(* CODESYS project ProjectX3_HLD.project

Project tree, tasks and I/O mapping:
  Device : CODESYS Control Win V3, 3S - Smart Software Solutions GmbH, version 3.5.16.20
    application Application
      libraries: Standard, * (System)
      task MainTask (cyclic, interval 20 ms, priority 1) calls Simulation, GAinstances, POLICY
      task VISU_TASK (cyclic, interval 100 ms, priority 31) calls VisuElems.Visu_Prg
      global variables GVL
      visualisation Visualization
      program Simulation [ST]
      function block DoorGA [SFC]: Init_active, READY_active, BUSY_active, Opening_active, Opening_exit, DONE1_active, Closing_active, Closing_exit, DONE_active, RESETDONE_active, Step1_active, Openit_exit, WAIT_1_exit, EverythingGood_active, OK_comunication_active, Init_timer_active, Comun_Problem_active
      function block CalculationGA [SFC]: READY_active, BUSY_active, Init_active, Current_active, Destination_active, VariableSet_active, VariableSet2_active, DoubleOutput_active, VariableSet_exit, DeckFault_active
      program POLICY [SFC]: Motor_ON_active, Motor_OFF_active, Velocity_I_exit, Motor_OFF_exit, Door_Open_active, Door_Open_exit, Door_Close_I_active, Door_Close_exit, Array_active, led_active, DeleteArray_active, Trans6, CalculationGA_active, MotorGA_exit, Velocity_I_active, Velocity_active, Calc_I_active, MotorGA_active, Init_active, Calc_I_exit, HLD_active, OK_comunication_2_active
      function block MotorGA [SFC]: motorON_active, motorOFF_active, BUSY_active, Trans0, READY_active, Motor_ON_I_active, Motor_OFF_I_active, Trans2, Init_active, DONE1_active, DONE2_active, DONE_active, RESETDONE_active
      function block VelocityGA [SFC]: Double_Output_active, MotorSlow_active, MotorSlow_exit, MotorFast_active, StopORGo_active, RampRange_active, Init_active, READY_active, BUSY_active, Vel_Init_active, Vel_Init_exit, Ramp_Fault_active
      program GAinstances [FBD]
  text list GlobalTextList
*)

// Device/Application/GVL
{attribute 'qualified_only'}
VAR_GLOBAL
	counting:INT;
	
(* Elevator managing variables*)
	Open: BOOL;				(* Sensor: the door is fully open*)
	Closed: BOOL;			(* Sensor: the door is fully closed*)
	LimitDown: BOOL;		(* Sensor: lower limit sensor, if TRUE the lift has reached the lower limit*)
	LimitUp: BOOL;			(* Sensor: upper limit sensor, if TRUE the lift has reached the upper limit*)
	DeckSensor: BOOL;		(* Sensor: if TRUE the cab is in proximity of a deck*)
	RampSensor: BOOL;		(* Sensor: if TRUE the cab is in proximity of a ramp*)
	Presence :BOOL; 		(* Sensor: if TRUE something blocks the door photocell*)
	Emergency: BOOL;		(* Input: if TRUE the emergency button has been pressed*)

	Closing: BOOL;			(* Actuator: if TRUE the door starts closing*)
	Opening: BOOL;			(* Actuator: the door starts opening*)
	Motor_on: BOOL;			(* Actuator: if TRUE the lift pulley motor start moving*)
	Up: BOOL;				(* Actuator parameter: if TRUE the lift moves upward, downward otherwise*)
	Vel: BOOL;				(* Actuator parameter: motor speed, if TRUE high speed, low speed otherwise*)


	Current: INT;
    Destination: INT;
	EmergencyVis: BOOL; 	(* Visualization: if TRUE the emergency light is turned on*)

	InitialDeck: INT := 1;	(* Only for simulation: variable used to define the initial deck*)
	InitCycle: BOOL := FALSE;(* Only for simulation: used to execute the instruction at the first cycle*)
	Height: INT;			(* Only for simulation: elevator height*)
	DeckRest: INT;        	(* Only for simulation: division rest for generating deck sensor*)
	Memory: INT;
	RampRest: INT;			(* Only for simulation: division rest for generating the ramp position*)
	MemoryR: INT;
	Door: INT;				(* Only for simulation: to visualize the closing of the door*)
	Displacement: INT;		(* Only for simulation: lift displacement, dependent on the motor speed*)

 (*Inputs: internal panel variables*)
	PG: BOOL;
	P1: BOOL;
	P2: BOOL;
	P3: BOOL;
	P4: BOOL;
	P5: BOOL;
	P6: BOOL;
	P7: BOOL;

(*Visualization: internal panel variables used to turn on the LED*)
	PGVis: BOOL;
	P1Vis: BOOL;
	P2Vis: BOOL;
	P3Vis: BOOL;
	P4Vis: BOOL;
	P5Vis: BOOL;
	P6Vis: BOOL;
	P7Vis: BOOL;

(*Inputs: external panel variables*)
	UpDeckG: BOOL;
	UpDeck1: BOOL;
	UpDeck2: BOOL;
	UpDeck3: BOOL;
	UpDeck4: BOOL;
	UpDeck5: BOOL;
	UpDeck6: BOOL;
	DownDeck7: BOOL;
	DownDeck6: BOOL;
	DownDeck5: BOOL;
	DownDeck4: BOOL;
	DownDeck3: BOOL;
	DownDeck2: BOOL;
	DownDeck1: BOOL;

(*Visualization: external panel variables used to turn on the LED*)
	UpDeckGVis: BOOL;
	UpDeck1Vis: BOOL;
	UpDeck2Vis: BOOL;
	UpDeck3Vis: BOOL;
	UpDeck4Vis: BOOL;
	UpDeck5Vis: BOOL;
	UpDeck6Vis: BOOL;
	DownDeck7Vis: BOOL;
	DownDeck6Vis: BOOL;
	DownDeck5Vis: BOOL;
	DownDeck4Vis: BOOL;
	DownDeck3Vis: BOOL;
	DownDeck2Vis: BOOL;
	DownDeck1Vis: BOOL;

(*Only for simulation: variables used to simulate the fault on deck sensor*)
	SensorG: BOOL;				(* if TRUE the magnetic information for deck G is lost and the deck sensor cannot become TRUE*)
	Sensor1: BOOL;				(* if TRUE the magnetic information for deck 1 is lost and the deck sensor cannot become TRUE*)
	Sensor2: BOOL;
	Sensor3: BOOL;
	Sensor4: BOOL;
	Sensor5: BOOL;
	Sensor6: BOOL;
	Sensor7: BOOL;
	FaultSensorAlarm: BOOL; 	(* Visulaization: if TRUE alerts the user of a deck sensor fault*)

(*Only for simulation: variables used to simulate the fault on ramp sensor*)
	RampGUp: BOOL;
	Ramp1Down: BOOL;
	Ramp1Up:BOOL;
	Ramp2Down: BOOL;
	Ramp2Up:BOOL;
	Ramp3Down: BOOL;
	Ramp3Up:BOOL;
	Ramp4Down: BOOL;
	Ramp4Up:BOOL;
	Ramp5Down: BOOL;
	Ramp5Up:BOOL;
	Ramp6Down: BOOL;
	Ramp6Up:BOOL;
	Ramp7Down: BOOL;
	FaultRampAlarm: BOOL; 		(* Visulaization: if TRUE alerts the user of a ramp sensor fault*)
	SensorGOK: BOOL;
	Sensor1OK: BOOL;
	Sensor2OK: BOOL;
	Sensor6OK: BOOL;
	Sensor3OK: BOOL;
	Sensor4OK: BOOL;
	Sensor5OK: BOOL;
	Sensor7OK: BOOL;
	RampGUpOK: BOOL;
	Ramp1DownOK: BOOL;
	Ramp1UpOK: BOOL;
	Ramp2DownOK: BOOL;
	Ramp2UpOK: BOOL;
	Ramp3DownOK: BOOL;
	Ramp3UpOK: BOOL;
	Ramp4DownOK: BOOL;
	Ramp4UpOK: BOOL;
	Ramp5DownOK: BOOL;
	Ramp5UpOK: BOOL;
	Ramp6DownOK: BOOL;
	Ramp6UpOK: BOOL;
	Ramp7DownOK: BOOL;
	Ramp7UpOK: BOOL;
	
	DoorGA_1: DoorGA;
	MotorGA_1: MotorGA;
	CalculationGA_1: CalculationGA;
	VelocityGA_1: VelocityGA;
	
	Vel_2: BOOL; //copy of the Value of Vel to use it in another GA
	go_up_2: BOOL; //copy of the Value of go_up to use it in another GA
	Motor_on_2: BOOL; //copy of the Value of Motor_on to use it in another GA (CalculationGA)
	DeckSensor_2:BOOL; //copy of the Value of DeckSensor to use it in another GA (VelocityGA)
	RampSensor_2:BOOL; //copy of the Value of RampSensor to use it in another GA (CalculationGA)
	Ramp_Range_2:BOOL; //this is the output value of the VelocityGA
	
	Broken1:INT; //output of CalculationGA
	End_Run:BOOL; //Allarm: if it is TRUE we have reached one of the two limit sensors
	
	A_up: ARRAY[0..7] OF BOOL;
	A_down: ARRAY[0..7] OF BOOL;
	L: ARRAY[0..7] OF BOOL;
	RampAlarm:BOOL;	
	
	HLD_global:TIME; //High Level Diagnostic variable
	Comunication_Missed:BOOL; //warning if we have a comunication problem btw GA and policy
	timerGA:TIME; //Value of timer.t passed as output from doorGA to be used in the policy
	init_timeGA:TIME; 
END_VAR

// Device/Application/Simulation
PROGRAM Simulation
VAR
END_VAR

(* Initial position of the cab inside the hoistway. It is executed only at the first cycle.  *)
IF NOT GVL.InitCycle THEN
			GVL.InitCycle := TRUE ;
			GVL.Height := 20 * GVL.InitialDeck;
		    GVL.Door := 0;
			GVL.Current := GVL.Height / 20;
END_IF;

(* Elevator management, these instructions are executed each cycle time*)

(* Elevator door control. *)
IF GVL.Closing THEN
	GVL.Door := GVL.Door + 1;		(*Closing door management*)
	GVL.Open := FALSE;
END_IF

IF GVL.Door >= 60 THEN						(* Closed door limit*)
	GVL.Closed := TRUE;
END_IF

IF GVL.Opening THEN
	GVL.Door := GVL.Door - 1; 	(* Opening door management*)
	GVL.Closed := FALSE;
END_IF

IF GVL.Door <= 0 THEN							(* Open door limit*)
	GVL.Open := TRUE;
END_IF


(* Maximum and minimum management in the door simulation*)
IF GVL.Door < 0 THEN
	 GVL.Door := 0;
END_IF

IF GVL.Door > 60 THEN
	GVL.Door := 60;
END_IF


(* Control of the cab position inside the hostway. *)
(* Displacement definition for graphic visualization*)
IF GVL.Vel THEN 
	GVL.Displacement := 2;
ELSE 
	GVL.Displacement := 1;
END_IF


(* Height modification relying on direction and speed*)
IF GVL.Motor_on AND GVL.Up THEN
	GVL.Height := GVL.Height + GVL.Displacement;
	GVL.LimitDown := FALSE;
END_IF

IF GVL.Motor_on AND NOT GVL.Up THEN
	GVL.Height := GVL.Height - GVL.Displacement;
	GVL.LimitUp := FALSE;
END_IF


(* Limits for visualization*)
IF GVL.Height < -20 THEN
	GVL.Height := -20;
END_IF

IF GVL.Height > 160 THEN
	GVL.Height := 160;
END_IF

(* Limit sensors management*)
IF GVL.Height <= -10 THEN
	GVL.LimitDown := TRUE;
END_IF

IF GVL.Height >= 150 THEN
	 GVL.LimitUp := TRUE;
END_IF


(*-------------------------------------------------------------------*)
(*  Fault Management (Deck and Ramp Sensors)   *)
(*-------------------------------------------------------------------*)
(* Deck Sensor*)
(* Range of value where the deck sensor is active*)
IF ((GVL.Height >= -1) AND (GVL.Height <= 1)) THEN
	GVL.SensorGOK := TRUE;
ELSE  
	GVL.SensorGOK := FALSE;
END_IF

IF ((GVL.Height >= 20-1) AND (GVL.Height <= 20+1)) THEN
	GVL.Sensor1OK := TRUE;
ELSE  
	GVL.Sensor1OK := FALSE;
END_IF

IF ((GVL.Height >= 40-1) AND (GVL.Height <= 40+1)) THEN
	GVL.Sensor2OK := TRUE;
ELSE  
	GVL.Sensor2OK := FALSE;
END_IF

IF ((GVL.Height >= 60-1) AND (GVL.Height <= 60+1)) THEN
	GVL.Sensor3OK := TRUE;
ELSE  
	GVL.Sensor3OK := FALSE;
END_IF

IF ((GVL.Height >= 80-1) AND (GVL.Height <= 80+1)) THEN
	GVL.Sensor4OK := TRUE;
ELSE  
	GVL.Sensor4OK := FALSE;
END_IF

IF ((GVL.Height >= 100-1) AND (GVL.Height <= 100+1)) THEN
	GVL.Sensor5OK := TRUE;
ELSE   
	GVL.Sensor5OK := FALSE;
END_IF

IF ((GVL.Height >= 120-1) AND (GVL.Height <= 120+1)) THEN
	GVL.Sensor6OK := TRUE;
ELSE  
	GVL.Sensor6OK := FALSE;
END_IF

IF ((GVL.Height >= 140-1) AND (GVL.Height <= 140+1)) THEN
	GVL.Sensor7OK := TRUE;
ELSE  
	GVL.Sensor7OK := FALSE;
END_IF

GVL.DeckSensor := (GVL.SensorGOK AND NOT GVL.SensorG) OR
				    (GVL.Sensor1OK AND NOT GVL.Sensor1) OR
				    (GVL.Sensor2OK AND NOT GVL.Sensor2) OR
				    (GVL.Sensor3OK AND NOT GVL.Sensor3) OR
				    (GVL.Sensor4OK AND NOT GVL.Sensor4) OR
				    (GVL.Sensor5OK AND NOT GVL.Sensor5) OR
				    (GVL.Sensor6OK AND NOT GVL.Sensor6) OR
				    (GVL.Sensor7OK AND NOT GVL.Sensor7);

(* Ramp Sensor*)
(* Range of value where the ramp sensor is active*)
IF ((GVL.Height >= 5-1) AND (GVL.Height <= 5+1)) THEN
	GVL.RampGUpOK := TRUE;
ELSE 
	GVL.RampGUpOK := FALSE;
END_IF

(* Ramp close to deck 1*)
IF ((GVL.Height >= 15-1) AND (GVL.Height <= 15+1)) THEN
	GVL.Ramp1DownOK := TRUE;
ELSE 
	GVL.Ramp1DownOK := FALSE;
END_IF

IF ((GVL.Height >= 25-1) AND (GVL.Height <= 25+1)) THEN
	GVL.Ramp1UpOK := TRUE;
ELSE 
	GVL.Ramp1UpOK := FALSE;
END_IF

(* Ramp close to deck 2*)
IF ((GVL.Height >= 35-1) AND (GVL.Height <= 35+1)) THEN
	GVL.Ramp2DownOK := TRUE;
ELSE 
	GVL.Ramp2DownOK := FALSE;
END_IF

IF ((GVL.Height >= 45-1) AND (GVL.Height <= 45+1)) THEN
	GVL.Ramp2UpOK := TRUE;
ELSE 
	GVL.Ramp2UpOK := FALSE;
END_IF

(*Ramp close to deck  3*)
IF ((GVL.Height >= 55-1) AND (GVL.Height <= 55+1)) THEN
	GVL.Ramp3DownOK := TRUE;
ELSE 
	GVL.Ramp3DownOK := FALSE;
END_IF

IF ((GVL.Height >= 65-1) AND (GVL.Height <= 65+1)) THEN
	GVL.Ramp3UpOK := TRUE;
ELSE 
	GVL.Ramp3UpOK := FALSE;
END_IF

(* Ramp close to deck  4*)
IF ((GVL.Height >= 75-1) AND (GVL.Height <= 75+1)) THEN
	GVL.Ramp4DownOK := TRUE;
ELSE 
	GVL.Ramp4DownOK := FALSE;
END_IF

IF ((GVL.Height >= 85-1) AND (GVL.Height <= 85+1)) THEN
	GVL.Ramp4UpOK := TRUE;
ELSE 
	GVL.Ramp4UpOK:=FALSE;
END_IF

(* Ramp close to deck  5*)
IF ((GVL.Height >= 95-1) AND (GVL.Height <= 95+1)) THEN
	GVL.Ramp5DownOK := TRUE;
ELSE 
	GVL.Ramp5DownOK := FALSE;
END_IF

IF ((GVL.Height >= 105-1) AND (GVL.Height <= 105+1)) THEN
	GVL.Ramp5UpOK := TRUE;
ELSE
	GVL.Ramp5UpOK := FALSE;
END_IF

(* Ramp close to deck  6*)
IF ((GVL.Height >= 115-1) AND (GVL.Height <= 115+1)) THEN
	GVL.Ramp6DownOK := TRUE;
ELSE 
	GVL.Ramp6DownOK := FALSE;
END_IF

IF ((GVL.Height >= 125-1) AND (GVL.Height <= 125+1)) THEN
	GVL.Ramp6UpOK := TRUE;
ELSE 
	GVL.Ramp6UpOK := FALSE;
END_IF

(* Ramp close to deck  7*)
IF ((GVL.Height >= 135-1) AND (GVL.Height <= 135+1)) THEN
	GVL.Ramp7DownOK := TRUE;
ELSE 
	GVL.Ramp7DownOK := FALSE;
END_IF

GVL.RampSensor:=(GVL.RampGUpOK AND NOT GVL.RampGUp) OR 
								(GVL.Ramp1DownOK AND NOT GVL.Ramp1Down ) OR 
								(GVL.Ramp1UpOK AND NOT GVL.Ramp1Up ) OR
								(GVL.Ramp2DownOK AND NOT GVL.Ramp2Down ) OR 
								(GVL.Ramp2UpOK AND NOT GVL.Ramp2Up ) OR
								(GVL.Ramp3DownOK AND NOT GVL.Ramp3Down ) OR
 								(GVL.Ramp3UpOK AND NOT GVL.Ramp3Up ) OR
								(GVL.Ramp4DownOK AND NOT GVL.Ramp4Down ) OR
 								(GVL.Ramp4UpOK AND NOT GVL.Ramp4Up ) OR
								(GVL.Ramp5DownOK AND NOT GVL.Ramp5Down ) OR
 								(GVL.Ramp5UpOK AND NOT GVL.Ramp5Up ) OR
								(GVL.Ramp6DownOK AND NOT GVL.Ramp6Down ) OR
								(GVL.Ramp6UpOK AND NOT GVL.Ramp6Up ) OR
								(GVL.Ramp7DownOK AND NOT GVL.Ramp7Down );

END_PROGRAM

// Device/Application/GAinstances
PROGRAM GAinstances
VAR
END_VAR

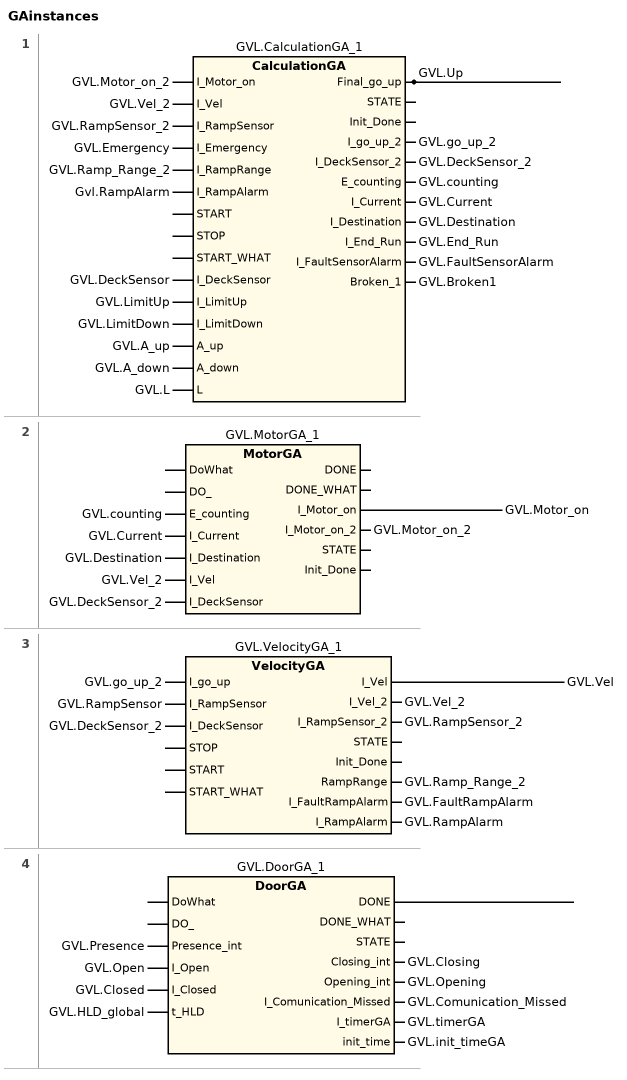
// NETWORK 1
GVL.CalculationGA_1(
    I_Motor_on := GVL.Motor_on_2,
    I_Vel := GVL.Vel_2,
    I_RampSensor := GVL.RampSensor_2,
    I_Emergency := GVL.Emergency,
    I_RampRange := GVL.Ramp_Range_2,
    I_RampAlarm := Gvl.RampAlarm,
    I_DeckSensor := GVL.DeckSensor,
    I_LimitUp := GVL.LimitUp,
    I_LimitDown := GVL.LimitDown,
    A_up := GVL.A_up,
    A_down := GVL.A_down,
    L := GVL.L,
    Final_go_up => GVL.Up,
    I_go_up_2 => GVL.go_up_2,
    I_DeckSensor_2 => GVL.DeckSensor_2,
    E_counting => GVL.counting,
    I_Current => GVL.Current,
    I_Destination => GVL.Destination,
    I_End_Run => GVL.End_Run,
    I_FaultSensorAlarm => GVL.FaultSensorAlarm,
    Broken_1 => GVL.Broken1); // CalculationGA

// NETWORK 2
GVL.MotorGA_1(
    E_counting := GVL.counting,
    I_Current := GVL.Current,
    I_Destination := GVL.Destination,
    I_Vel := GVL.Vel_2,
    I_DeckSensor := GVL.DeckSensor_2,
    I_Motor_on_2 => GVL.Motor_on_2); // MotorGA
GVL.Motor_on := GVL.MotorGA_1.I_Motor_on;

// NETWORK 3
GVL.VelocityGA_1(
    I_go_up := GVL.go_up_2,
    I_RampSensor := GVL.RampSensor,
    I_DeckSensor := GVL.DeckSensor_2,
    I_Vel_2 => GVL.Vel_2,
    I_RampSensor_2 => GVL.RampSensor_2,
    RampRange => GVL.Ramp_Range_2,
    I_FaultRampAlarm => GVL.FaultRampAlarm,
    I_RampAlarm => GVL.RampAlarm); // VelocityGA
GVL.Vel := GVL.VelocityGA_1.I_Vel;

// NETWORK 4
GVL.DoorGA_1(
    Presence_int := GVL.Presence,
    I_Open := GVL.Open,
    I_Closed := GVL.Closed,
    t_HLD := GVL.HLD_global,
    Closing_int => GVL.Closing,
    Opening_int => GVL.Opening,
    I_Comunication_Missed => GVL.Comunication_Missed,
    I_timerGA => GVL.timerGA,
    init_time => GVL.init_timeGA); // DoorGA

END_PROGRAM

// Device/Application/CalculationGA
FUNCTION_BLOCK CalculationGA
VAR_INPUT
	I_Motor_on:BOOL; //associated to Motor_on_2 from the policy
	I_Vel:BOOL; //associated to Vel_2 from the policy
	I_RampSensor:BOOL; //associated to RampSensor_2 from the policy
	
	I_Emergency:BOOL; //Variable associated to the button in the lift
	I_RampRange:BOOL; //Variable determinated in VelocityGA
	I_RampAlarm:BOOL; //Variable calculated in VelocityGA
	START: BOOL;
	STOP:BOOL;
	START_WHAT: STRING;
	I_DeckSensor: BOOL; //Sensor
	I_LimitUp:BOOL; //Sensor
	I_LimitDown: BOOL; //Sensor
	
	A_up: ARRAY[0..7] OF BOOL; //Array from the policy
	A_down: ARRAY[0..7] OF BOOL; //Array from the policy
	L: ARRAY[0..7] OF BOOL; //Array from the policy
	
	
END_VAR

VAR_OUTPUT
	Final_go_up:BOOL; //parameter associated to the real actuator UP
	STATE:STRING;
	Init_Done: BOOL; //this is useful to comunicate to the policy when the initialization is completed
	I_go_up_2:BOOL; //copy of the Value of go_up to use it in another GA
	I_DeckSensor_2:BOOL; //copy of the Value of I_DeckSensor to use it in another GA (MotorGA)
	E_counting:INT; //Variable explained in the Destination block
	I_Current:INT;
	I_Destination:INT;
	I_End_Run:BOOL; //Allarm if we reach one of the two limit sensors

	I_FaultSensorAlarm:BOOL; //variable associated to the LED of the interface 
	Broken_1:INT; //This variable store the information of the Broken DeckSensor
END_VAR

VAR	
	i:INT; //index used in the Destination block
	EndInit:BOOL;
	pippo:BOOL; //Variable used in the Current block
	FOUND:BOOL;	//Variable used in the Destination block
	FOUND_2:BOOL; //Variable used in the Destination block		
	//NET:BOOL; actually this variable is not used anymore, see the Destination block
	RampRange:BOOL;
	Temp_Destination:INT; //Variable used in the Destination block
	go_up:BOOL; //Variable used in the Destination block
	count_ramp:INT; //Variable used in the DeckFault block
	NRST:BOOL; //NRST stands for Not Ramp Sensor Twice, used in the DeckFault block
	NRST_2:BOOL; //NRST stands for Not Ramp Sensor Twice, used in the DeckFault block
	FOUND3:BOOL; //Variable used in the DeckFault block
END_VAR

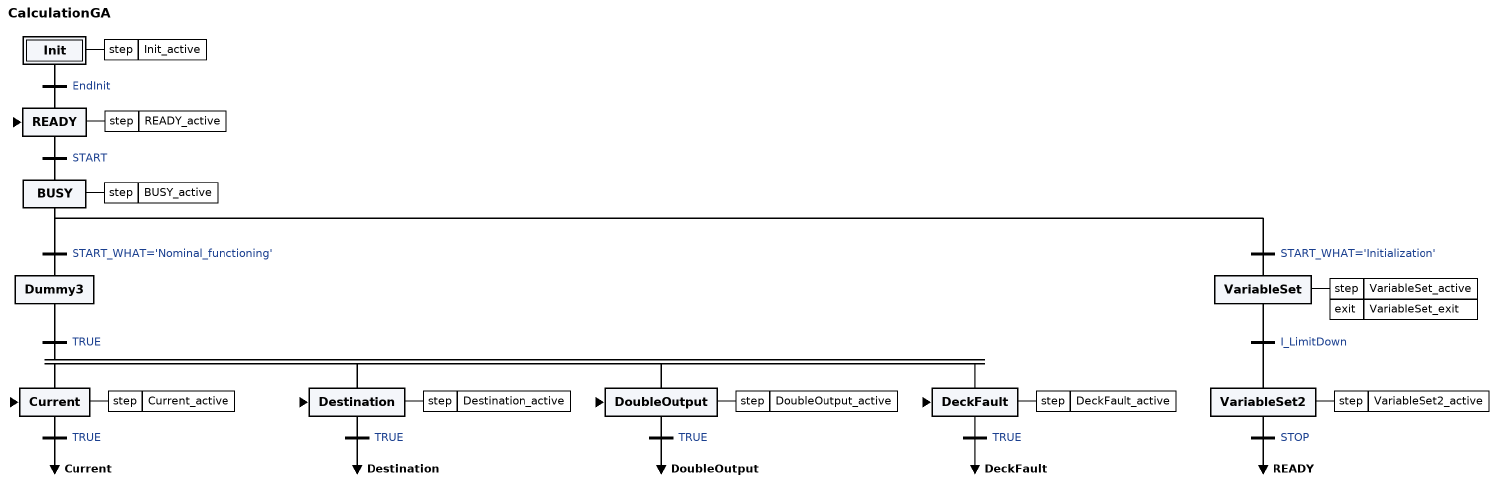
INITIAL_STEP Init:
    Init_active(N);  // step action
END_STEP
TRANSITION FROM Init TO READY
    := EndInit;
END_TRANSITION
STEP READY:
    READY_active(N);  // step action
END_STEP
TRANSITION FROM READY TO BUSY
    := START;
END_TRANSITION
STEP BUSY:
    BUSY_active(N);  // step action
END_STEP
TRANSITION FROM BUSY TO Dummy3
    := START_WHAT='Nominal_functioning';
END_TRANSITION
STEP Dummy3:
END_STEP
TRANSITION FROM Dummy3 TO (Current, Destination, DoubleOutput, DeckFault)
    := TRUE;
END_TRANSITION
STEP Current:
    Current_active(N);  // step action
END_STEP
STEP Destination:
    Destination_active(N);  // step action
END_STEP
TRANSITION FROM Destination TO Destination
    := TRUE;
END_TRANSITION
STEP DoubleOutput:
    DoubleOutput_active(N);  // step action
END_STEP
TRANSITION FROM DoubleOutput TO DoubleOutput
    := TRUE;
END_TRANSITION
STEP DeckFault:
    DeckFault_active(N);  // step action
END_STEP
TRANSITION FROM DeckFault TO DeckFault
    := TRUE;
END_TRANSITION
TRANSITION FROM Current TO Current
    := TRUE;
END_TRANSITION
TRANSITION FROM BUSY TO VariableSet
    := START_WHAT='Initialization';
END_TRANSITION
STEP VariableSet:
    VariableSet_active(N);  // step action
    VariableSet_exit(P0);  // exit action
END_STEP
TRANSITION FROM VariableSet TO VariableSet2
    := I_LimitDown;
END_TRANSITION
STEP VariableSet2:
    VariableSet2_active(N);  // step action
END_STEP
TRANSITION FROM VariableSet2 TO READY
    := STOP;
END_TRANSITION

ACTION READY_active:
STATE:='READY';
END_ACTION

ACTION BUSY_active:
STATE:='BUSY';
END_ACTION

ACTION Init_active:
STATE:='Init';
I_Current:=0; //Initially we set I_Current:=0, this does not matter a lot as in the block VariableSet2 we will
//initialized it properly 
EndInit:=TRUE;
END_ACTION

ACTION Current_active:
//This block calculates the Current floor.
//It changes the GVL.Current value when the GVL.DeckSensor turns ON(+1 if we are going up, -1 otherwise).
//
//We implent the variable pippo because the turning on of the decksensor can last more then a PLC cycle(we don't know the duration
//of the signal), so thanks to pippo we can avoid counting twice the change of GVL.Current value.

IF I_DeckSensor THEN
	IF pippo=TRUE THEN
		IF go_up THEN
			I_Current:=I_Current + 1;
		ELSE 
			I_Current:=I_Current - 1;
		END_IF
		pippo:=FALSE;
	END_IF
END_IF
IF I_DeckSensor=FALSE THEN
	pippo:=TRUE;
END_IF
END_ACTION

ACTION Destination_active:
(*The goal of destination is to calculate the next stop.

The priority of the elevator is determined as follow:
1. If the lift is going up the priority is given to all the calls coming from a floor higher than the current position of the lift:
	1.1. The updeck and inside button calls in a increasing array index order (from the lower to the higher floor)
	1.2. The downdeck calls in a decreasing array index order (from the higher to the lower floor)

2. If the lift is going down the priority is given to all the calls coming from a floor lower than the current position of the lift:
	2.1. The downdeck and inside button calls in a decreasing array index order (from the higher to the lower floor)
	2.2. The updeck calls in a increasing array index order (from the lower to the higher floor)*)


FOUND:=FALSE; //This variable has two goals: the first is to change the direction of go_up if it is FALSE, in this way
//the code start checking for calls from a lower floor; the second is to skip the checking of the downdeck (updeck calls),
//if the lift is going up (going down)
FOUND_2:=FALSE; (*The objective of this variable is to avoid the update of Temp_Destination with a call that actually has
a lower priority*)

IF go_up=TRUE THEN
	FOR i:=(I_Current+1) TO 7 BY 1 DO
		IF (A_up[i]=TRUE OR L[i]=TRUE) AND FOUND_2=FALSE THEN 
			  Temp_Destination:=i;
			  FOUND:=TRUE;
			  FOUND_2:=TRUE;
		END_IF
	END_FOR
	
	
	IF FOUND=FALSE THEN
		FOR i:= 7 TO (I_Current+1) BY -1 DO
			IF A_down[i]=TRUE AND FOUND_2=FALSE THEN 
			  Temp_Destination:=i;
			  FOUND:=TRUE;
			  FOUND_2:=TRUE;
			END_IF
		END_FOR
	END_IF
	IF FOUND=FALSE THEN
		go_up:=FALSE;
	END_IF
END_IF


IF go_up=FALSE THEN
	FOR i:=(I_Current-1) TO 0 BY -1 DO
		IF (A_down[i]=TRUE OR L[i]=TRUE) AND FOUND_2=FALSE THEN 
			  Temp_Destination:=i;
			  FOUND:=TRUE;
			  FOUND_2:=TRUE;
		END_IF
	END_FOR
	
	IF FOUND=FALSE THEN
		FOR i:= 0 TO (I_Current-1) BY 1 DO
			IF A_up[i]=TRUE AND FOUND_2=FALSE THEN 
			  Temp_Destination:=i;
			  FOUND:=TRUE;
			  FOUND_2:=TRUE;
			 END_IF
		END_FOR
	END_IF
	
	IF FOUND=FALSE THEN
		go_up:=TRUE ;
		Temp_Destination:=I_Current; //if there are no calls from any floors than we set the destination 
		//equal to the current floor as we are already in the final position
	END_IF
END_IF

(*THE FOLLOWING COMMENT IS AN UNUSED CODE, WRITTEN THINKING THAT THE BEHAVIOR OF THE EMERGENCY BUTTON WAS EQUAL TO THE OTHER
BUTTONS. DUE TO THIS MISINTERPRETATION WE USED E_COUNTING INSTEAD OF I_EMERGENCY AS VARIABLE TO REFER TO A PRESS OF THE 
BUTTON.
WE DECIDE TO NOT ELIMINATE E_COUNTING BECAUSE CAN BE HELPFUL TO HAVE A CODE THAT COULD ALSO WORK WITH ANOTHER TYPOLOGY OF 
BUTTON*)

(*//NET stands for NOT_EMERGENCY_TWICE, E_counting stands for EMERGENCY_counting
//The following lines uses two new variables: NET to avoid counting twice the emergency button if this is long
//pressed; E_counting to memorize how many times is actually pressed the emergency button (E_counting=0 nominal
//functioning and E_counting=1 emergency)
IF I_Emergency=TRUE AND NET=FALSE THEN 
	NET:=TRUE;
	E_counting:=E_counting+1;
	IF E_counting=2 THEN //when Emergency is pressed for the second time, we have to go back to the nominal functioning setting E_counting:=0 
		E_counting:=0;
	END_IF
END_IF
//when emergency is realised also NET gets false
IF I_Emergency=FALSE THEN
	NET:=FALSE;
END_IF*)

IF I_Emergency=TRUE THEN
	E_counting:=1;
ELSE 
	E_counting:=0;
END_IF

//If we are in emergency, we need to update Temp_Destination with the first next floor (according to the direction of the lift).
//But if the elevator is not in condition to slow down on time for the next floor then I_Destination will be not update 
//with the value of Temp_Destination thanks to the algorithm at line 129.
IF E_counting=1 AND I_Motor_on=TRUE THEN
	IF go_up=TRUE THEN
		Temp_Destination:=I_Current+1;
	ELSE Temp_Destination:=I_Current-1;
	END_IF
END_IF

(*This code is related to the DeckSensor Fault. When this problem happens we are not able to stop the elevator at the
problematic floor, so once that we determinated the broken DeckSensor thanks to Broken_1, if the destination was 
exactly that floor then we update Temp_Destination according to go_up with the next floor. This is not true when 
Broken_1=0 or Broken_1=7, as in this case no next floor exits. For this two cases the problem is solved in the Policy
in the block Array*)
IF Broken_1=Temp_Destination AND Broken_1<>7 AND Broken_1<>0 THEN
	IF go_up THEN
		Temp_Destination:=Broken_1+1;
	ELSE
		Temp_Destination:=Broken_1-1;
	END_IF
END_IF



//We update the I_Destination value (variable corresponding to the real next destination) with the Temp_Destination 
//value calculated with the above priorities. The variable Temp_Destination does not keep in consideration the current 
//velocity of the lift.
// As we cannot stop the lift if the elevetor is going fast, the I_Destination value update happens only if the lift is 
//out of the RampRange or it is still at a floor (motor off).
IF I_RampRange=FALSE OR I_Motor_on=FALSE THEN
	I_Destination:=Temp_Destination;
END_IF

(*When the LimitUp Sensor is reached, this can happen only if the 7th DeckSensor is broken, then we need to change the value
of both Final_go_up and go_up. Moreover we set TRUE I_End_Run that it is used in the Policy in the Array block*)
IF I_LimitUp=TRUE THEN
	I_End_Run:=TRUE;
	Final_go_up:=FALSE;
	go_up:=FALSE;
END_IF

(*When the LimitDown Sensor is reached, this can happen only if the Ground DeckSensor is broken, then we need to change 
the value of both Final_go_up and go_up. Moreover we set TRUE I_End_Run that it is used in the Policy in the Array block*)
IF I_LimitDown=TRUE THEN
	I_End_Run:=TRUE;
	Final_go_up:=TRUE;
	go_up:=TRUE;
END_IF

//I_End_Run stays TRUE only when one of the two Limit Sensor is TRUE
IF I_LimitDown=FALSE AND I_LimitUp=FALSE THEN
	I_End_Run:=FALSE;
END_IF

IF I_RampAlarm THEN
	IF GVL.Current=0 THEN
		Final_go_up:=TRUE;
		go_up:=TRUE;
	ELSIF GVL.Current=7 THEN
		Final_go_up:=FALSE;
		go_up:=FALSE;
	END_IF
END_IF


//go_up is a variable that is update in every moment, whereas Final_go_up is update only if the motor is OFF. This
//because the change of direction can happen only when we are still. Moreover if this is not done, there are problems
//because the UP actuator changes its direction before stopping, causing a misalignment when it stops at a floor. 
//To avoid some troubles of priority when we have multiple calls and a RampAlarm, it is useful to allow the lift 
//to change direction also in case of a RampAlarm, because it could be necessary to service first a call coming from
//the opposite direction
IF I_Motor_on=FALSE OR I_RampAlarm THEN
	Final_go_up:=go_up;
END_IF
END_ACTION

ACTION VariableSet_active:
//In this phase many variables are initializated, especially we set Final_go_up as false because we need 
//to bring the elevator to the bottom first

pippo:=FALSE;
Final_go_up:=FALSE;
i:=0;
FOUND:=FALSE;

//NET:=FALSE; Variable not used anymore. See Destionation Block
E_counting:=0;

Init_Done:=TRUE; //comunication to the policy
END_ACTION

ACTION VariableSet2_active:
//In this phase many variables are initializated, especially we set Final_go_up as TRUE because we need 
//to bring the elevator to the first floor
Final_go_up:=TRUE;
//copy of the Value of Final_go_up to use it in the policy
I_go_up_2:=Final_go_up;

I_Current:=-1; //The starting value is -1 because I_Current increases its value for each DeckSensor and 
//before reaching the first floor the elevator will meet the Ground DeckSensor and the 1st floor DeckSensor

Broken_1:=8; //As this variable store the information of the Broken DeckSensor, we choose this  starting
//value because no floor 8 exits, so its like saying that all the sensors are working

NRST:=FALSE;
NRST_2:=FALSE;
FOUND3:=FALSE;

Init_Done:=TRUE; //comunication with the policy
END_ACTION

ACTION DoubleOutput_active:
//This two operation are done to copy the value of Final_go_up and I_DeckSensor into two new variables in order
//two use this value in another GA without violated the rules of the GA approach

//copy of the Value of go_up to use it in another GA
I_go_up_2:=Final_go_up;

//copy of the Value of go_up to use it in another GA
I_DeckSensor_2:=I_DeckSensor;
END_ACTION

ACTION VariableSet_exit:
Init_Done:=FALSE;
END_ACTION

ACTION DeckFault_active:
//A possible broken DeckSensor is managed thanks to this block. If a DeckSensor is broken the lift
//keeps working but it cannot serve any call coming from the floor where the DeckSensor is broken.
//The detection is done counting the number of RampSensors met without meeting a DeckSensor; if this count
//reaches three we have a broken DeckSensor.

//NRST and NRST_2 are used to count I_RampSensor only once when it is activated. The initial values for NRST 
//and NRST_2 are FALSE.

//Whenever I_RampSensor becomes TRUE, NRST is set as TRUE. This is excuted only for the first cycle for which
//I_RampSensor is TRUE because possible double counting of the same signal are stopped by NRST_2, that some 
//lines down is set as TRUE.
IF I_RampSensor AND NRST_2=FALSE THEN
	NRST:=TRUE; //NRST stands for Not Ramp Sensor Twice
END_IF

//When I_RampSensor gets FALSE we reset the values of NRST and NRST_2 to be ready for the next time in which
//I_RampSensor becomes TRUE.
IF I_RampSensor=FALSE THEN
	NRST:=FALSE;
	NRST_2:=FALSE;
END_IF

//When we have detected the first turning TRUE of I_RampSensor, we have NRST=TRUE, so we update the variable
//count_ramp. This variable keeps the count of how many ramp sensors are met without meeting a DeckSensor.
//This little block is excuted only once per meeting with a RampSensor, indeed the first time we excute it we also 
//set NRST_2:=TRUE and NRST:=FALSE; this will block the first IF of this code as well as this IF itself. We can 
//excute again this two IF only after a reset of NRST and NRST_2, that happens when I_RampSensor gets FALSE.
IF NRST THEN 
	count_ramp:=count_ramp+1;
	NRST_2:=TRUE;
	NRST:=FALSE; 
END_IF
 
//If a DeckSensor is met count_ramp can be reset to 0. A warning is given only if count_ramp reaches 3.
IF I_DeckSensor THEN 
	count_ramp:=0;
	FOUND3:=FALSE; //This variable, that here is reset, it necessary to execute the next IF only once if 
				  //count_ramp reaches 3, otherwise the value of Broken_1 and I_Current would be updated to many
				  //times.
END_IF

(*When count_ramp reaches 3 AND we are AT the first cycle OF THIS situation (that means: FOUND3:=FALSE), THEN 
we want to give an allarm of broken DeckSensor. Moreover to ensure the correct fuctioning of the elevator
we have to force the update of the Current Position as usually this is achieved thanks to the DeckSensor.
We also store the information of which DeckSensor (in the variable Broken_1) is broken in order to use it
in the policy in the block DeleteArray where we manage the cancellation of the calls.
The two operation just mentioned are done also according to the value of Final_go_up.
Particular cases are those in which the broken DeckSensor belongs either to the Ground floor or to the 7th floor,
in these cases the detection is done thanks to the LimitUp and LimitDown sensor.*)
IF (count_ramp=3 OR I_LimitUp OR I_LimitDown) AND FOUND3=FALSE THEN
	I_FaultSensorAlarm:=TRUE;
	IF Final_go_up AND (I_LimitUp=FALSE AND I_LimitDown=FALSE) THEN
		Broken_1:=I_Current+1;
		I_Current:=I_Current+1;
	ELSIF Final_go_up=FALSE AND (I_LimitUp=FALSE AND I_LimitDown=FALSE) THEN
		Broken_1:=I_Current-1;
		I_Current:=I_Current-1;
	ELSIF I_LimitUp=TRUE THEN
		Broken_1:=I_Current+1;
		I_Current:=I_Current+1;
	ELSIF I_LimitDown=TRUE THEN
		Broken_1:=I_Current-1;
		I_Current:=I_Current-1;		
	END_IF
	FOUND3:=TRUE; //We set it to TRUE to avoid to excute this block again. Actually when a new DeckSensor is 
				  //reached, FOUND3 gets FALSE again, but at that point count_ramp is reset to zero, so we 
				  //do not have problems.
END_IF
END_ACTION

END_FUNCTION_BLOCK

// Device/Application/POLICY

PROGRAM POLICY
VAR
	OperationOK:BOOL; //variable used in the DO-DONE GAs
	Synchronisation:BOOL; //variable used in the DO-DONE GAs
	EndInit: BOOL;
	
	P_Comunication_Missed:BOOL;
END_VAR

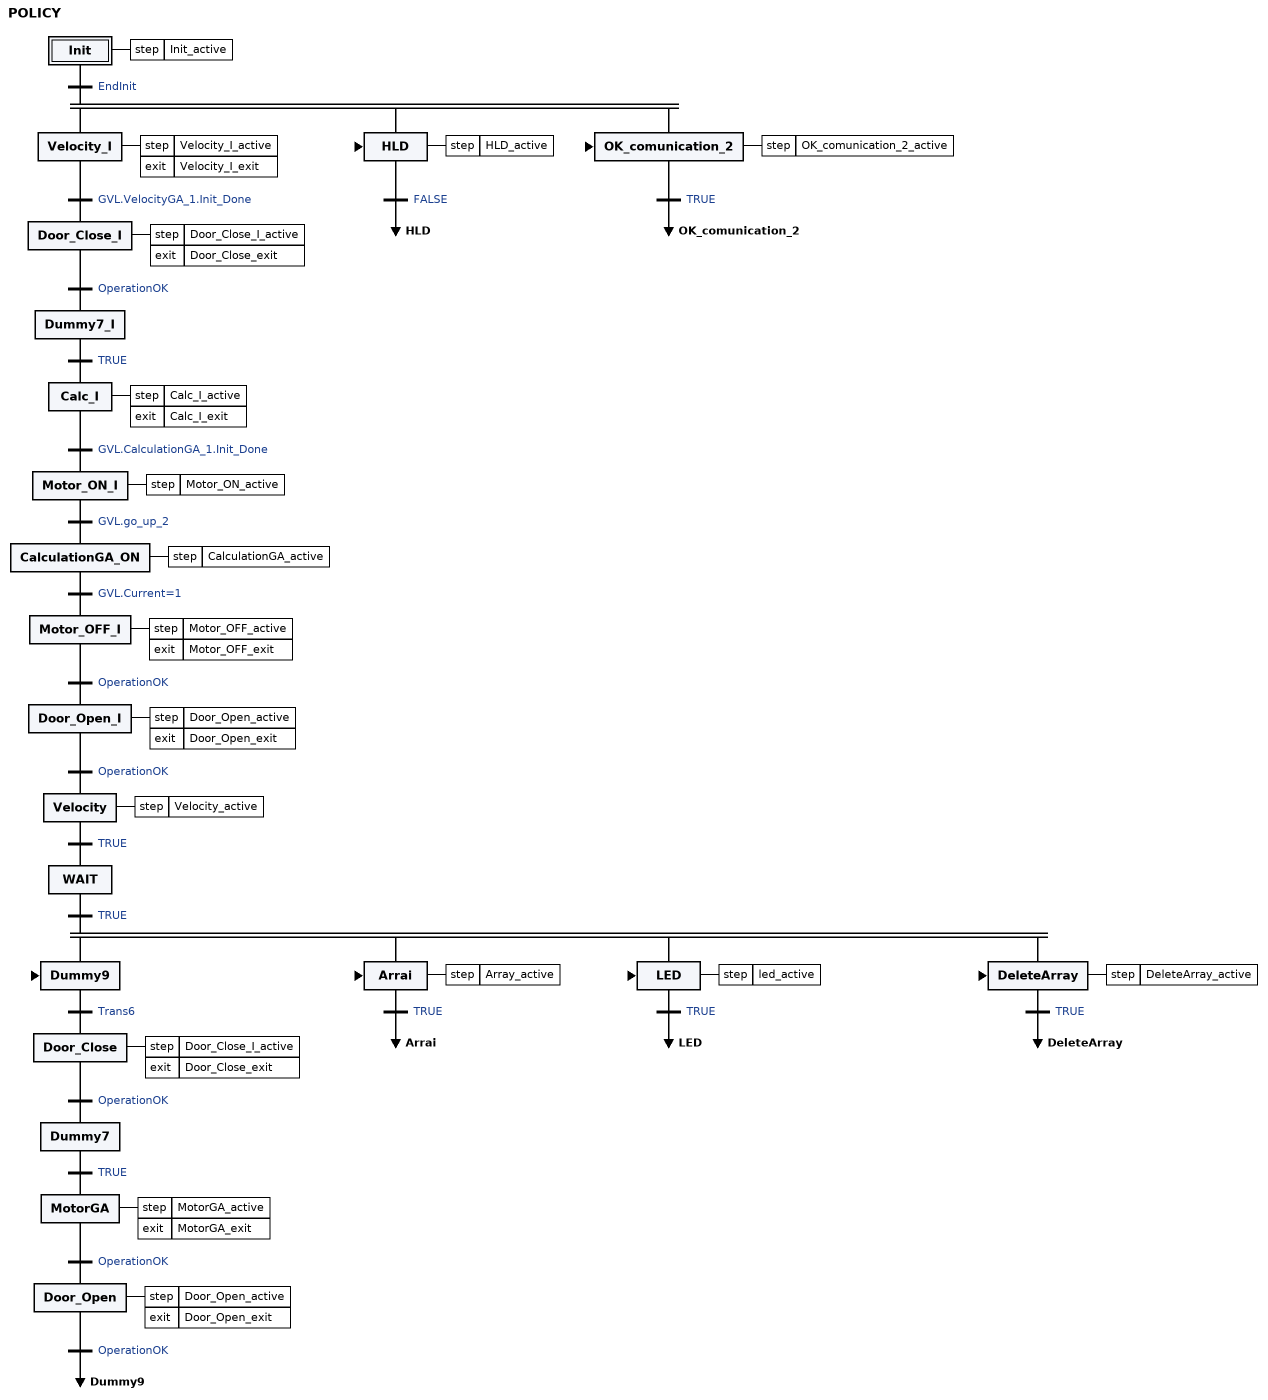
INITIAL_STEP Init:
    Init_active(N);  // step action
END_STEP
TRANSITION FROM Init TO (Velocity_I, HLD, OK_comunication_2)
    := EndInit;
END_TRANSITION
STEP Velocity_I:
    Velocity_I_active(N);  // step action
    Velocity_I_exit(P0);  // exit action
END_STEP
STEP HLD:
    HLD_active(N);  // step action
END_STEP
TRANSITION FROM HLD TO HLD
    := FALSE;
END_TRANSITION
STEP OK_comunication_2:
    OK_comunication_2_active(N);  // step action
END_STEP
TRANSITION FROM OK_comunication_2 TO OK_comunication_2
    := TRUE;
END_TRANSITION
TRANSITION FROM Velocity_I TO Door_Close_I
    := GVL.VelocityGA_1.Init_Done;
END_TRANSITION
STEP Door_Close_I:
    Door_Close_I_active(N);  // step action
    Door_Close_exit(P0);  // exit action
END_STEP
TRANSITION FROM Door_Close_I TO Dummy7_I
    := OperationOK;
END_TRANSITION
STEP Dummy7_I:
END_STEP
TRANSITION FROM Dummy7_I TO Calc_I
    := TRUE;
END_TRANSITION
STEP Calc_I:
    Calc_I_active(N);  // step action
    Calc_I_exit(P0);  // exit action
END_STEP
TRANSITION FROM Calc_I TO Motor_ON_I
    := GVL.CalculationGA_1.Init_Done;
END_TRANSITION
STEP Motor_ON_I:
    Motor_ON_active(N);  // step action
END_STEP
TRANSITION FROM Motor_ON_I TO CalculationGA_ON
    := GVL.go_up_2;
END_TRANSITION
STEP CalculationGA_ON:
    CalculationGA_active(N);  // step action
END_STEP
TRANSITION FROM CalculationGA_ON TO Motor_OFF_I
    := GVL.Current=1;
END_TRANSITION
STEP Motor_OFF_I:
    Motor_OFF_active(N);  // step action
    Motor_OFF_exit(P0);  // exit action
END_STEP
TRANSITION FROM Motor_OFF_I TO Door_Open_I
    := OperationOK;
END_TRANSITION
STEP Door_Open_I:
    Door_Open_active(N);  // step action
    Door_Open_exit(P0);  // exit action
END_STEP
TRANSITION FROM Door_Open_I TO Velocity
    := OperationOK;
END_TRANSITION
STEP Velocity:
    Velocity_active(N);  // step action
END_STEP
TRANSITION FROM Velocity TO WAIT
    := TRUE;
END_TRANSITION
STEP WAIT:
END_STEP
TRANSITION FROM WAIT TO (Dummy9, Arrai, LED, DeleteArray)
    := TRUE;
END_TRANSITION
STEP Dummy9:
END_STEP
TRANSITION FROM Dummy9 TO Door_Close
    := Trans6;
END_TRANSITION
STEP Door_Close:
    Door_Close_I_active(N);  // step action
    Door_Close_exit(P0);  // exit action
END_STEP
TRANSITION FROM Door_Close TO Dummy7
    := OperationOK;
END_TRANSITION
STEP Dummy7:
END_STEP
TRANSITION FROM Dummy7 TO MotorGA
    := TRUE;
END_TRANSITION
STEP MotorGA:
    MotorGA_active(N);  // step action
    MotorGA_exit(P0);  // exit action
END_STEP
TRANSITION FROM MotorGA TO Door_Open
    := OperationOK;
END_TRANSITION
STEP Door_Open:
    Door_Open_active(N);  // step action
    Door_Open_exit(P0);  // exit action
END_STEP
TRANSITION FROM Door_Open TO Dummy9
    := OperationOK;
END_TRANSITION
STEP Arrai:
    Array_active(N);  // step action
END_STEP
TRANSITION FROM Arrai TO Arrai
    := TRUE;
END_TRANSITION
STEP LED:
    led_active(N);  // step action
END_STEP
TRANSITION FROM LED TO LED
    := TRUE;
END_TRANSITION
STEP DeleteArray:
    DeleteArray_active(N);  // step action
END_STEP
TRANSITION FROM DeleteArray TO DeleteArray
    := TRUE;
END_TRANSITION

ACTION Motor_ON_active:
//The 4th GA called by the  policy is MotorGA. Also here it is ask to the GA to performe some steps useful for
//the initialization of the elevator. Indeed the motor is turned on, and the GA keep working even if the policy
//at a certain point goes over. The Initialization process of this GA ends after the block Motor_OFF_I (see later)

IF  GVL.MotorGA_1.STATE ='READY'  THEN
	GVL.MotorGA_1.DO_:=TRUE;
	GVL.MotorGA_1.DoWhat:='Init1';
END_IF
END_ACTION

ACTION Motor_OFF_active:
//MotorGA actually is already active, indeed what we do here is just understand if the initialization of this
//GA is DONE, this would mean that the motor is now OFF as we reached the first floor
IF  GVL.MotorGA_1.STATE='BUSY' AND GVL.MotorGA_1.DONE THEN
	GVL.MotorGA_1.DO_:=FALSE;
	Synchronisation:=TRUE;
END_IF

OperationOK:=Synchronisation AND NOT GVL.MotorGA_1.DONE;
END_ACTION

ACTION Velocity_I_exit:
IF  GVL.VelocityGA_1.STATE='BUSY' THEN
	GVL.VelocityGA_1.START:=FALSE;
	GVL.VelocityGA_1.STOP:=TRUE;
END_IF
END_ACTION

ACTION Motor_OFF_exit:
Synchronisation:=FALSE;
OperationOK:=FALSE;
END_ACTION

ACTION Door_Open_active:
//Now that we have reached correctly the first floor to end the initialization, we open the doors.

//This action is associated to two different blocks of the POLICY:
//1. Door_Open_I
//2. Door_Open
//this because the DoorGA must be called without any difference when we are doing the
//Initialization and during the nominal_functioning



IF  GVL.DoorGA_1.STATE='READY'  THEN
	GVL.DoorGA_1.DO_:=TRUE;
	GVL.DoorGA_1.DoWhat:='Open';
END_IF

IF  GVL.DoorGA_1.STATE='BUSY' AND GVL.DoorGA_1.DONE THEN
	GVL.DoorGA_1.DO_:=FALSE;
	Synchronisation:=TRUE;
END_IF

OperationOK:=Synchronisation AND NOT GVL.DoorGA_1.DONE;
END_ACTION

ACTION Door_Open_exit:
Synchronisation:=FALSE;
OperationOK:=FALSE;
END_ACTION

ACTION Door_Close_I_active:
//Once that VelocityGA has done with its Initialization we can call DoorGA to close the doors

//This action is associated to two different blocks of the POLICY:
//1. Door_Close_I
//2. Door_Close
//this because the DoorGA must be called without any difference when we are doing the
//Initialization and during the nominal_functioning

IF  GVL.DoorGA_1.STATE ='READY'  THEN
	GVL.DoorGA_1.DO_:=TRUE;
	GVL.DoorGA_1.DoWhat:='Close';
END_IF

IF  GVL.DoorGA_1.STATE='BUSY' AND GVL.DoorGA_1.DONE THEN
	GVL.DoorGA_1.DO_:=FALSE;
	Synchronisation:=TRUE;
END_IF

OperationOK:=Synchronisation AND NOT GVL.DoorGA_1.DONE;
END_ACTION

ACTION Door_Close_exit:
Synchronisation:=FALSE;
OperationOK:=FALSE;
END_ACTION

ACTION Array_active:
// We use 3 arrays to register the button signal (UpDeck,DownDeck and internal buttons) in order to maintain the signal
//during the time. 
// If a button is pushed twice the value of the array is not affected.
IF GVL.UpDeckG=TRUE THEN
	GVL.A_up[0]:=1;
END_IF
IF GVL.UpDeck1=TRUE THEN
	GVL.A_up[1]:=1;
END_IF
IF GVL.UpDeck2=TRUE THEN
	GVL.A_up[2]:=1;
END_IF
IF GVL.UpDeck3=TRUE THEN
	GVL.A_up[3]:=1;
END_IF
IF GVL.UpDeck4=TRUE THEN
	GVL.A_up[4]:=1;
END_IF
IF GVL.UpDeck5=TRUE THEN
	GVL.A_up[5]:=1;
END_IF
IF GVL.UpDeck6=TRUE THEN
	GVL.A_up[6]:=1;
END_IF
GVL.A_up[7]:=0;



IF GVL.DownDeck1=TRUE THEN
	GVL.A_down[1]:=1;
END_IF
IF GVL.DownDeck2=TRUE THEN
	GVL.A_down[2]:=1;
END_IF
IF GVL.DownDeck3=TRUE THEN
	GVL.A_down[3]:=1;
END_IF
IF GVL.DownDeck4=TRUE THEN
	GVL.A_down[4]:=1;
END_IF
IF GVL.DownDeck5=TRUE THEN
	GVL.A_down[5]:=1;
END_IF
IF GVL.DownDeck6=TRUE THEN
	GVL.A_down[6]:=1;
END_IF
IF GVL.DownDeck7=TRUE THEN
	GVL.A_down[7]:=1;
END_IF
GVL.A_down[0]:=0;


IF GVL.PG=TRUE THEN
	GVL.L[0]:=1;
END_IF
IF GVL.P1=TRUE THEN
	GVL.L[1]:=1;
END_IF
IF GVL.P2=TRUE THEN
	GVL.L[2]:=1;
END_IF
IF GVL.P3=TRUE THEN
	GVL.L[3]:=1;
END_IF
IF GVL.P4=TRUE THEN
	GVL.L[4]:=1;
END_IF
IF GVL.P5=TRUE THEN
	GVL.L[5]:=1;
END_IF
IF GVL.P6=TRUE THEN
	GVL.L[6]:=1;
END_IF
IF GVL.P7=TRUE THEN
	GVL.L[7]:=1;
END_IF


//When the FaultSensorAlarm is TRUE menas that a DeckSensor is broken. If End_Run is true means that the elevator
//has reached either the LimitUp Sensor or the LimitDown Sensor and one of this two is still TRUE.
//So when both of this situation are prensent means that the DeckSensor of the 7th floor or of the Ground Floor
//is broken. To check which of the two sensor is broken we have just to understand approximately where is the
//Elevator, so we can say that Current>5 then for sure the broken DeckSensor is the one of the 7th floor, 
//otherwise is the one of the Ground floor. According to this we can decide to force a call from the nearest
//floor to stop the elevator there.
IF GVL.FaultSensorAlarm AND GVL.End_Run THEN
	IF GVL.Current>5 THEN
		GVL.L[6]:=1;
	ELSE
		GVL.L[1]:=1;
	END_IF
END_IF

(*These last lines of code are executed when we have a fault with a RampSensor. When this is detected, by a 
dedicated block in the VelocityGA, then we need to dissimulate some calls to stop correctly the lift. Basically 
if the ramp sensor of the ground floor or of the seventh floor is broken we send the elevator to the 2st floor
or to 5th floor. The elevator is not sent to the 1st or to the 6th just because also these floors are affected 
if the ramp sensor of the Ground or of the 7th floor is broken (1st floor is not avaiable if we are coming from
Ground whereas is avaiable if we are coming from the 2nd, similar thing for the 6th*)
IF GVL.RampAlarm THEN
	IF GVL.Current=0 THEN
		 GVL.L[2]:=1;
	ELSIF GVL.Current=7 THEN
		 GVL.L[5]:=1;
	END_IF
END_IF

(*For all the other broken ramp sensors if the destination is at the floor where we intend to stop, then a fake
call from the above or under floor, according to the direction of the lift, is done (we don't actually use the 
variable destination because this is updated when we become aware of the fault and so some calculation can be wrong.
To avoid these problem we just check if there were calls from the problematic floor*)
IF GVL.RampAlarm AND GVL.Destination<>0 AND GVL.Destination<>7 THEN
	IF GVL.go_up_2 THEN
		IF GVL.L[GVL.Current] OR GVL.A_up[GVL.Current] OR GVL.A_down[GVL.Current] THEN
			GVL.L[GVL.Current+1]:=1;
		END_IF
	ELSE 
		IF GVL.L[GVL.Current] OR GVL.A_up[GVL.Current] OR GVL.A_down[GVL.Current] THEN
			GVL.L[GVL.Current-1]:=1;
		END_IF
	END_IF
END_IF
END_ACTION

ACTION led_active:
//Turning on the right LED is achieved just copying the value of the arrays in the Vis variables	
	GVL.PGVis:=GVL.L[0];
	GVL.P1Vis:=GVL.L[1];
	GVL.P2Vis:=GVL.L[2];
	GVL.P3Vis:=GVL.L[3];
	GVL.P4Vis:=GVL.L[4];
	GVL.P5Vis:=GVL.L[5];
	GVL.P6Vis:=GVL.L[6];
	GVL.P7Vis:=GVL.L[7];
	GVL.UpDeckGVis:=GVL.A_up[0];
	GVL.UpDeck1Vis:=GVL.A_up[1];
	GVL.UpDeck2Vis:=GVL.A_up[2];
	GVL.UpDeck3Vis:=GVL.A_up[3];
	GVL.UpDeck4Vis:=GVL.A_up[4];
	GVL.UpDeck5Vis:=GVL.A_up[5];
	GVL.UpDeck6Vis:=GVL.A_up[6];
	GVL.DownDeck1Vis:=GVL.A_down[1];
	GVL.DownDeck2Vis:=GVL.A_down[2];
	GVL.DownDeck3Vis:=GVL.A_down[3];
	GVL.DownDeck4Vis:=GVL.A_down[4];
	GVL.DownDeck5Vis:=GVL.A_down[5];
	GVL.DownDeck6Vis:=GVL.A_down[6];
	GVL.DownDeck7Vis:=GVL.A_down[7];

//The Emergency LED is turned on according to the value of GVL.counting, a variable that actually as the 
//same value of GVL.Emergency (see Destinatione in the CalculationGA to understand why)
	IF GVL.counting=1 THEN
		GVL.EmergencyVis:=TRUE;
	ELSE
		GVL.EmergencyVis:=FALSE;
	END_IF
END_ACTION

ACTION DeleteArray_active:
//Thanks to this block we eliminate the values stored in the arrays if the lift has reached the right floor (and so the users' call
//is satisfied).
//
//Every time the lift arrives to a floor we eliminate: 
//1. always the array value of the button inside the lift corresponding to the current floor
//2. the array Updeck/Downdeck value corresponding to the current floor if the lift is going Up/Down.

IF GVL.Motor_on=FALSE THEN
	GVL.L[GVL.Current]:=FALSE;
	IF GVL.Up=TRUE THEN
		GVL.A_up[GVL.Current]:=FALSE;
	ELSE GVL.A_down[GVL.Current]:=FALSE;
	END_IF
END_IF

//When a Deck Sensor is broken we cannot serve that floor, so all the calls coming from the unavailable floor
//(indentified by GVL.Broken1) are immediately deleted.
IF GVL.FaultSensorAlarm THEN
	GVL.L[GVL.Broken1]:=FALSE;
	GVL.A_up[GVL.Broken1]:=FALSE;
	GVL.A_down[GVL.Broken1]:=FALSE;
END_IF


(*This part is helpful to delete the call from the groud floor and the 7th floor when their RampSensor is broken, as 
we cannot stop there going fast*)
IF GVL.RampAlarm THEN
	IF GVL.Current=0 THEN
		 GVL.L[0]:=FALSE;
		 GVL.A_up[0]:=FALSE;
		 
	ELSIF GVL.Current=7 THEN
		GVL.L[7]:=FALSE;
		GVL.A_down[7]:=FALSE;
	END_IF
END_IF


(*To avoid main complex problem related to the motion direction in relation to the active call, we decide to delete, 
if present a call coming from the floor immediately before (if UP is TRUE) of the floor where the Ramp Fault is
detected (mirrored thing if we are going down ). This is a little throwback.*)
IF GVL.RampAlarm THEN
	IF GVL.go_up_2 THEN
		IF GVL.Current<>0 THEN (*this is need because otherwise when the ground ramp sensor is broken, this code is 
			excuted when the direction is changed to reach the 2nd floor*)
			GVL.L[GVL.Current-1]:=FALSE;
			GVL.A_down[GVL.Current-1]:=FALSE;
			GVL.A_up[GVL.Current-1]:=FALSE;
		END_IF
	ELSE 
		IF GVL.Current<>7 THEN (*this is need because otherwise when the 7th floor ramp sensor is broken, this code is 
			excuted when the direction is changed to reach the 5th floor*)
			GVL.L[GVL.Current+1]:=FALSE;
			GVL.A_down[GVL.Current+1]:=FALSE;
			GVL.A_up[GVL.Current+1]:=FALSE;
		END_IF
	END_IF
END_IF
END_ACTION

TRANSITION Trans6:
//GVL.counting is the global variable for E_counting

//The doors can be closed only if we are not in emergency and during the nominal functioning we need to close them
//only if the calculated current position is different from the calculated destination. The same condition can be 
//found inside the motorGA to start the Motor. This because we close the doors only if then we move the lift (so the
//motor will be started).
GVL.counting<>1 AND GVL.Current<>GVL.Destination
END_TRANSITION

ACTION CalculationGA_active:
//Once that the Initialization of CalculationGA is done we can recall the same GA asking for  Nominal_functioning.
//It is important to call this GA because we need to start counting the value of Current as the next transition
//depends on it
IF  GVL.CalculationGA_1.STATE='READY' THEN
	GVL.CalculationGA_1.START:=TRUE;
	GVL.CalculationGA_1.STOP:=FALSE;
	GVL.CalculationGA_1.START_WHAT:='Nominal_functioning';
END_IF
END_ACTION

ACTION MotorGA_exit:
Synchronisation:=FALSE;
OperationOK:=FALSE;
END_ACTION

ACTION Velocity_I_active:
//The policy immediadely call the  VelocityGA asking for the Initialization procedure. In this way we are 
//sure to operate with LOW SPEED
IF  GVL.VelocityGA_1.STATE='READY' THEN
	GVL.VelocityGA_1.START:=TRUE;
	GVL.VelocityGA_1.STOP:=FALSE;
	GVL.VelocityGA_1.START_WHAT:='Initialization';
END_IF
END_ACTION

ACTION Velocity_active:
//Here the initialization is finished, so we can call VelocityGA and start it in its Nominal_functioning. This
//GA will continue working as long as the elevator works. 

IF  GVL.VelocityGA_1.STATE='READY' THEN
	GVL.VelocityGA_1.START:=TRUE;
	GVL.VelocityGA_1.STOP:=FALSE;
	GVL.VelocityGA_1.START_WHAT:='Nominal_functioning';
END_IF
END_ACTION

ACTION Calc_I_active:
//Now we call CalculationGA whose Variable Initialization is divided in two parts. This is the first part, where some 
//important variables are initializated; especially we set UP as FALSE because we need to bring the elevator
//to the bottom first

IF  GVL.CalculationGA_1.STATE='READY' THEN
	GVL.CalculationGA_1.START:=TRUE;
	GVL.CalculationGA_1.STOP:=FALSE;
	GVL.CalculationGA_1.START_WHAT:='Initialization';
END_IF

//When the second part of the varible initialization takes place (this happens whene the lift meets LimitDown)
//in CalculationGA other variables are initializated;
//especially Current is set to -1 as we will meet 2 deck sensors going to the 1st floor. Moreover also the value
//of UP is changed as now we need to go up
END_ACTION

ACTION MotorGA_active:
//When we call MotorGA, it will perform two main actions: turn the motor ON to reach the destination, then 
//turn it OFF giving the signal of DONE to the policy

IF  GVL.MotorGA_1.STATE ='READY'  THEN
	GVL.MotorGA_1.DO_:=TRUE;
	GVL.MotorGA_1.DoWhat:='Nominal_fuctioning';
END_IF

IF  GVL.MotorGA_1.STATE='BUSY' AND GVL.MotorGA_1.DONE THEN
	GVL.MotorGA_1.DO_:=FALSE;
	Synchronisation:=TRUE;
END_IF

OperationOK:=Synchronisation AND NOT GVL.MotorGA_1.DONE;
END_ACTION

ACTION Init_active:
//some variables are initializated as intended just to ensure the correct functioning of the code 

GVL.FaultRampAlarm:=FALSE;
GVL.FaultSensorAlarm:=FALSE;

EndInit:=TRUE;
END_ACTION

ACTION Calc_I_exit:
IF  GVL.CalculationGA_1.STATE='BUSY' THEN
	GVL.CalculationGA_1.STOP:=TRUE;
	GVL.CalculationGA_1.START:=FALSE;
END_IF
END_ACTION

ACTION HLD_active:
GVL.HLD_global:=HLD.t;
END_ACTION

ACTION OK_comunication_2_active:
(*As P_Init_Time store the difference between the two times, then this equation, if the comunication works
 properly at each cycle should be FALSE. But if the comunication is delayed or missed then we got a warning*)

IF HLD.t>GVL.timerGA+GVL.init_timeGA THEN
	P_Comunication_Missed:=TRUE;
END_IF
END_ACTION

END_PROGRAM

// Device/Application/MotorGA
FUNCTION_BLOCK MotorGA
VAR_INPUT
	DoWhat: STRING;
	DO_: BOOL;
	E_counting: INT; //Variable determinated in CalculationGA
	I_Current:INT; //Variable determinated in CalculationGA
	I_Destination:INT; //Variable determinated in CalculationGA
	I_Vel: BOOL; //associated to Vel_2 from the policy
	I_DeckSensor: BOOL;//Sensor
	
END_VAR

VAR_OUTPUT
	DONE:BOOL;
	DONE_WHAT:STRING;
	I_Motor_on: BOOL; //Actuator
	I_Motor_on_2: BOOL; //copy of the Value of I_Motor_on to use it in another GA (CalculationGA)
	STATE: STRING;
	Init_Done: BOOL;
	
END_VAR

VAR
	EndInit:BOOL;
END_VAR

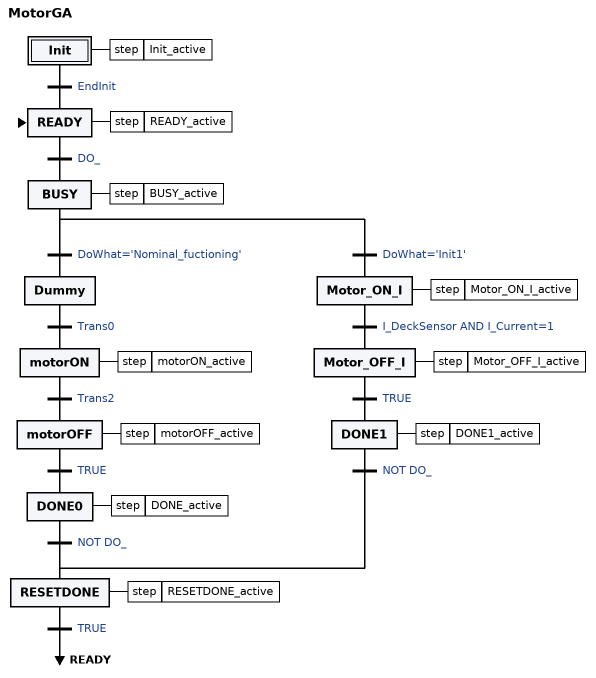
INITIAL_STEP Init:
    Init_active(N);  // step action
END_STEP
TRANSITION FROM Init TO READY
    := EndInit;
END_TRANSITION
STEP READY:
    READY_active(N);  // step action
END_STEP
TRANSITION FROM READY TO BUSY
    := DO_;
END_TRANSITION
STEP BUSY:
    BUSY_active(N);  // step action
END_STEP
TRANSITION FROM BUSY TO Dummy
    := DoWhat='Nominal_fuctioning';
END_TRANSITION
STEP Dummy:
END_STEP
TRANSITION FROM Dummy TO motorON
    := Trans0;
END_TRANSITION
STEP motorON:
    motorON_active(N);  // step action
END_STEP
TRANSITION FROM motorON TO motorOFF
    := Trans2;
END_TRANSITION
STEP motorOFF:
    motorOFF_active(N);  // step action
END_STEP
TRANSITION FROM motorOFF TO DONE0
    := TRUE;
END_TRANSITION
STEP DONE0:
    DONE_active(N);  // step action
END_STEP
TRANSITION FROM DONE0 TO RESETDONE
    := NOT DO_;
END_TRANSITION
TRANSITION FROM BUSY TO Motor_ON_I
    := DoWhat='Init1';
END_TRANSITION
STEP Motor_ON_I:
    Motor_ON_I_active(N);  // step action
END_STEP
TRANSITION FROM Motor_ON_I TO Motor_OFF_I
    := I_DeckSensor AND I_Current=1;
END_TRANSITION
STEP Motor_OFF_I:
    Motor_OFF_I_active(N);  // step action
END_STEP
TRANSITION FROM Motor_OFF_I TO DONE1
    := TRUE;
END_TRANSITION
STEP DONE1:
    DONE1_active(N);  // step action
END_STEP
TRANSITION FROM DONE1 TO RESETDONE
    := NOT DO_;
END_TRANSITION
STEP RESETDONE:
    RESETDONE_active(N);  // step action
END_STEP
TRANSITION FROM RESETDONE TO READY
    := TRUE;
END_TRANSITION

ACTION motorON_active:
I_Motor_on:=TRUE;

//copy of the Value of I_Motor_on to use it in another GA (CalculationGA)
I_Motor_on_2:=I_Motor_on;
END_ACTION

ACTION motorOFF_active:
I_Motor_on:=FALSE;

//copy of the Value of I_Motor_on to use it in another GA (CalculationGA)
I_Motor_on_2:=I_Motor_on;
END_ACTION

ACTION BUSY_active:
STATE:='BUSY';
END_ACTION

TRANSITION Trans0:
//GVL.counting is the global variable for E_counting

//The motor can be turned ON only if we are not in emergency (be careful, this does not mean that whenever the button 
//emergency is pressed the motor goes off) and during the normal functioning we need to turn ON the motor to move the lift
//only if the calculated current position is different from the calculated destination
E_counting<>1 AND I_Current<>I_Destination
END_TRANSITION

ACTION READY_active:
STATE:= 'READY';
END_ACTION

ACTION Motor_ON_I_active:
//When the policy needs the motor in turned ON for the initialization and we stop it we reach the first floor
I_Motor_on:=TRUE;

//copy of the Value of I_Motor_on to use it in another GA (CalculationGA)
I_Motor_on_2:=I_Motor_on;
END_ACTION

ACTION Motor_OFF_I_active:
//When the first floor is reached we immediately stop the motor
I_Motor_on:=FALSE;

//copy of the Value of I_Motor_on to use it in another GA (CalculationGA)
I_Motor_on_2:=I_Motor_on;
END_ACTION

TRANSITION Trans2:
//GVL.counting is the global variable for E_counting

(*The motor is turned OFF in two situations, both valid only if the velocity is slow and decksensor is TRUE:
	1. The current position equates the destination 
	2. The 'E_counting' is equal to 1 and so we are in emergency. In this case the point 1 could fail because, 
		as soon the new decksensor is reached, the Destination Block, that is still working considering the emergency
	 	mood(E_counting=1), calculates a new temp_destination = GVL.Current + 1, even if actually we need to stop now.*)
(I_Current=I_Destination AND I_Vel=FALSE AND I_DeckSensor) OR (E_counting=1 AND I_Vel=FALSE AND I_DeckSensor)
END_TRANSITION

ACTION Init_active:
STATE:='Init';
EndInit:=TRUE;
END_ACTION

ACTION DONE1_active:
//Comunication to the policy
DONE:=TRUE;
DONE_WHAT:='Init1';
END_ACTION

ACTION DONE2_active:
DONE:=TRUE;
DONE_WHAT:='Init2';
END_ACTION

ACTION DONE_active:
//Comunication to the policy
DONE:=TRUE;
DONE_WHAT:='Nominal_fuctioning';
END_ACTION

ACTION RESETDONE_active:
DONE:=FALSE;
END_ACTION

END_FUNCTION_BLOCK

// Device/Application/DoorGA
FUNCTION_BLOCK DoorGA
VAR_INPUT
	DoWhat: STRING;
	DO_: BOOL;
	Presence_int: BOOL; //Sensor
	I_Open:BOOL; //Sensor
	I_Closed:BOOL; //Sensor
	
	t_HLD:TIME; //Variable to be sure of to do not miss comunications from the policy
END_VAR
VAR_OUTPUT
	DONE:BOOL;
	DONE_WHAT:STRING;
	STATE:STRING;
	Closing_int: BOOL; //Actuator
	Opening_int: BOOL; //Actuator
	
	I_Comunication_Missed:BOOL; //variable to comunicate a problem in the comunication with the 
	//policy
	I_timerGA:TIME; //this is the value of timer.t set as output for the policy
	init_time:TIME; //variable used for the HLD, that memorize the initial difference between
	//the timer of the GA and the timer of the Policy
END_VAR
VAR
	EndInit:BOOL;
	EverythingGood:BOOL; //this variable is helpful to start the closing of the doors 
	//again when it is interrupted because presence was true
	
	PLCcycle:TIME; //duration of a PLC cycle
END_VAR

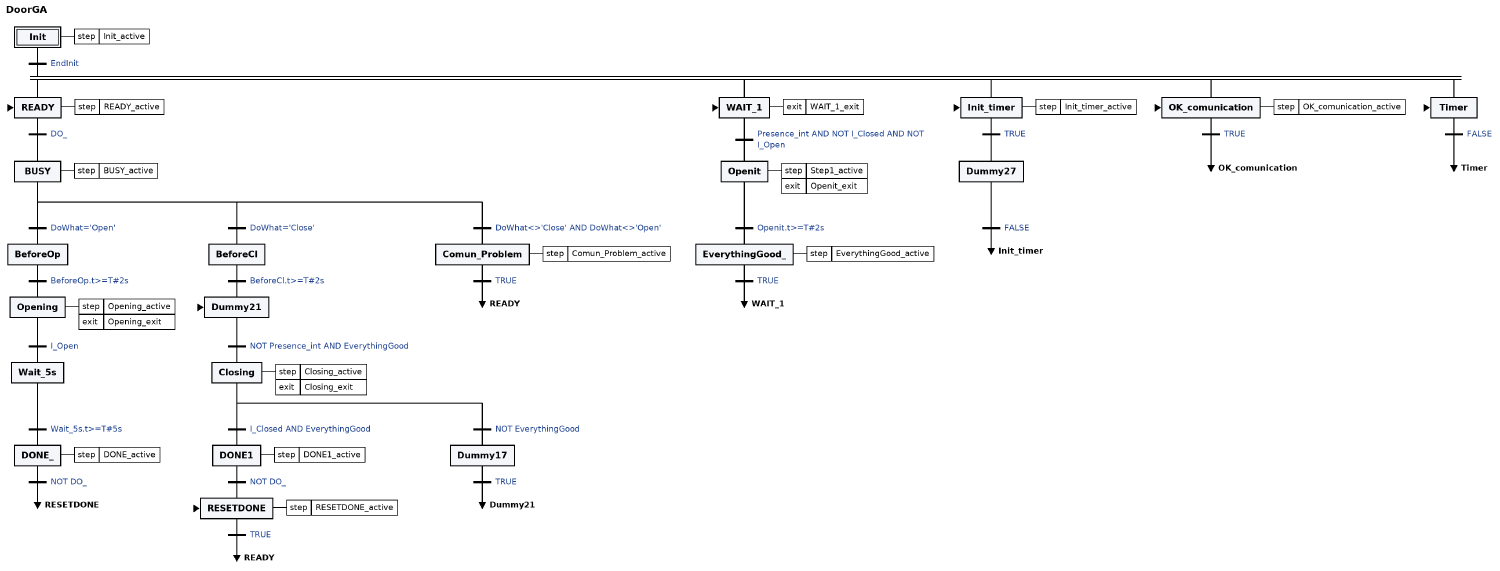
INITIAL_STEP Init:
    Init_active(N);  // step action
END_STEP
TRANSITION FROM Init TO (READY, WAIT_1, Init_timer, OK_comunication, Timer)
    := EndInit;
END_TRANSITION
STEP READY:
    READY_active(N);  // step action
END_STEP
STEP WAIT_1:
    WAIT_1_exit(P0);  // exit action
END_STEP
TRANSITION FROM WAIT_1 TO Openit
    := Presence_int AND NOT I_Closed AND NOT I_Open;
END_TRANSITION
STEP Openit:
    Step1_active(N);  // step action
    Openit_exit(P0);  // exit action
END_STEP
TRANSITION FROM Openit TO EverythingGood_
    := Openit.t>=T#2s;
END_TRANSITION
STEP EverythingGood_:
    EverythingGood_active(N);  // step action
END_STEP
TRANSITION FROM EverythingGood_ TO WAIT_1
    := TRUE;
END_TRANSITION
STEP Init_timer:
    Init_timer_active(N);  // step action
END_STEP
TRANSITION FROM Init_timer TO Dummy27
    := TRUE;
END_TRANSITION
STEP Dummy27:
END_STEP
TRANSITION FROM Dummy27 TO Init_timer
    := FALSE;
END_TRANSITION
STEP OK_comunication:
    OK_comunication_active(N);  // step action
END_STEP
TRANSITION FROM OK_comunication TO OK_comunication
    := TRUE;
END_TRANSITION
STEP Timer:
END_STEP
TRANSITION FROM Timer TO Timer
    := FALSE;
END_TRANSITION
TRANSITION FROM READY TO BUSY
    := DO_;
END_TRANSITION
STEP BUSY:
    BUSY_active(N);  // step action
END_STEP
TRANSITION FROM BUSY TO BeforeOp
    := DoWhat='Open';
END_TRANSITION
STEP BeforeOp:
END_STEP
TRANSITION FROM BeforeOp TO Opening
    := BeforeOp.t>=T#2s;
END_TRANSITION
STEP Opening:
    Opening_active(N);  // step action
    Opening_exit(P0);  // exit action
END_STEP
TRANSITION FROM Opening TO Wait_5s
    := I_Open;
END_TRANSITION
STEP Wait_5s:
END_STEP
TRANSITION FROM Wait_5s TO DONE_
    := Wait_5s.t>=T#5s;
END_TRANSITION
STEP DONE_:
    DONE_active(N);  // step action
END_STEP
TRANSITION FROM DONE_ TO RESETDONE
    := NOT DO_;
END_TRANSITION
TRANSITION FROM BUSY TO BeforeCl
    := DoWhat='Close';
END_TRANSITION
STEP BeforeCl:
END_STEP
TRANSITION FROM BeforeCl TO Dummy21
    := BeforeCl.t>=T#2s;
END_TRANSITION
STEP Dummy21:
END_STEP
TRANSITION FROM Dummy21 TO Closing
    := NOT Presence_int AND EverythingGood;
END_TRANSITION
TRANSITION FROM BUSY TO Comun_Problem
    := DoWhat<>'Close' AND DoWhat<>'Open';
END_TRANSITION
STEP Comun_Problem:
    Comun_Problem_active(N);  // step action
END_STEP
TRANSITION FROM Comun_Problem TO READY
    := TRUE;
END_TRANSITION
STEP Closing:
    Closing_active(N);  // step action
    Closing_exit(P0);  // exit action
END_STEP
TRANSITION FROM Closing TO DONE1
    := I_Closed AND EverythingGood;
END_TRANSITION
STEP DONE1:
    DONE1_active(N);  // step action
END_STEP
TRANSITION FROM DONE1 TO RESETDONE
    := NOT DO_;
END_TRANSITION
STEP RESETDONE:
    RESETDONE_active(N);  // step action
END_STEP
TRANSITION FROM Closing TO Dummy17
    := NOT EverythingGood;
END_TRANSITION
STEP Dummy17:
END_STEP
TRANSITION FROM Dummy17 TO Dummy21
    := TRUE;
END_TRANSITION
TRANSITION FROM RESETDONE TO READY
    := TRUE;
END_TRANSITION

ACTION Init_active:
STATE:='Init';

EverythingGood:=TRUE; //if TRUE no problem with presence for the moment
PLCcycle:=T#21MS;
I_Comunication_Missed:=FALSE;//used for HLD

EndInit:=TRUE;
END_ACTION

ACTION READY_active:
STATE:='READY';
END_ACTION

ACTION BUSY_active:
STATE:='BUSY';
END_ACTION

ACTION Opening_active:
Opening_int:=TRUE;
END_ACTION

ACTION Opening_exit:
//Once the action is completed we can turn OFF the actuator
Opening_int:=FALSE;
END_ACTION

ACTION DONE1_active:
//Comunication to the policy
DONE:=TRUE;
DONE_WHAT:='Close';
END_ACTION

ACTION Closing_active:
//If the presence is  actived when the action is not completed yet, the value of Closing_int is set as
//false thanks to the parallelism seen at the beginnig of the DoorGA

Closing_int:=TRUE;
END_ACTION

ACTION Closing_exit:
//Once the action is completed we can turn OFF the actuator
Closing_int:=FALSE;
END_ACTION

ACTION DONE_active:
//Comunication to the policy
DONE:=TRUE;
DONE_WHAT:='Open';
END_ACTION

ACTION RESETDONE_active:
DONE:=FALSE;
END_ACTION

ACTION Step1_active:
//Thanks to this parallelism, whenever presence becomes true the closing procedure is interrupted and and
//the opening takes place.

Closing_int:=FALSE;
Opening_int:=TRUE;
END_ACTION

ACTION Openit_exit:
Opening_int:=FALSE;
END_ACTION

ACTION WAIT_1_exit:
EverythingGood:=FALSE; //as soon as presence gets TRUE, EverythingGood changes its value
END_ACTION

ACTION EverythingGood_active:
EverythingGood:=TRUE; //The door are open again EverythingGood is set again to TRUE. If the presence sensor
//is still activeted then we will re-execute this branch again and again
END_ACTION

ACTION OK_comunication_active:
(*As init_time store the difference between the two times, then this equation, if the comunication works
 properly at each cycle should be FALSE. But if the comunication is delayed or missed then we got a warning*)

IF init_time+timer.t>t_HLD+PLCcycle THEN //Note that t_HLD is always delaye buy one PLC cycle
	I_Comunication_Missed:=TRUE;
END_IF

//copy the value to use it as output
I_timerGA:=timer.t;
END_ACTION

ACTION Init_timer_active:
//init_time store the difference between the two times

init_time:=t_HLD;
END_ACTION

ACTION Comun_Problem_active:
I_Comunication_Missed:=TRUE;
END_ACTION

END_FUNCTION_BLOCK

// Device/Application/VelocityGA
FUNCTION_BLOCK VelocityGA
VAR_INPUT
	I_go_up: BOOL; //associated to go_up_2 from the policy
	I_RampSensor: BOOL; //Sensor
	I_DeckSensor:BOOL; //associated to DeckSensor_2 from the policy
	STOP: BOOL;	
	START: BOOL;
	START_WHAT: STRING;
END_VAR
VAR_OUTPUT
	I_Vel:BOOL; //Actuator
	I_Vel_2:BOOL; //copy of the Value of I_Vel to use it in another GA
	I_RampSensor_2: BOOL; //copy of the Value of I_RampSensor to use it in another GA
	STATE: STRING;
	Init_Done: BOOL; //it comunicates to the policy that the initialization is completed
	RampRange:BOOL; //This variable is used to understand if the elevator is inside two RampSensor or not:
					//it is considered inside (RampRange=TRUE) if the elevator is between the two ramp sensor
					//of the same floor.
	I_FaultRampAlarm:BOOL; //Comunication with the policy
	I_RampAlarm:BOOL; //Comunication with the policy
END_VAR
VAR
	minni:BOOL; //its task is explained in the block StopORGo 
	pluto:BOOL; //its task is explained in the block Ramp_Range
	bunny:BOOL; //its task is explained in the block StopORGo
	count_ramp:INT;
	NRST:BOOL; //NRST stands for Not Ramp Sensor Twice
	NRST_2:BOOL;
	pip:BOOL; //its task is explained in the block Ramp_Fault
	EndInit:BOOL;
END_VAR

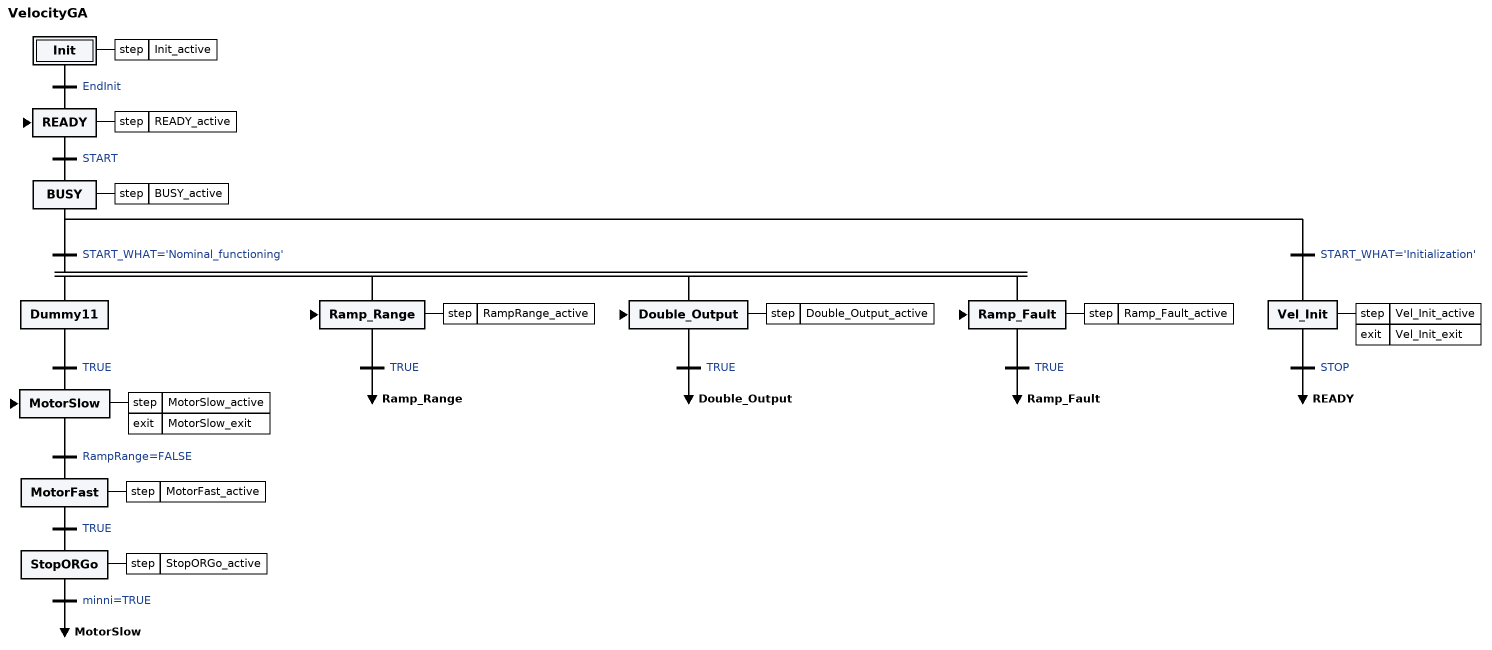
INITIAL_STEP Init:
    Init_active(N);  // step action
END_STEP
TRANSITION FROM Init TO READY
    := EndInit;
END_TRANSITION
STEP READY:
    READY_active(N);  // step action
END_STEP
TRANSITION FROM READY TO BUSY
    := START;
END_TRANSITION
STEP BUSY:
    BUSY_active(N);  // step action
END_STEP
TRANSITION FROM BUSY TO (Dummy11, Ramp_Range, Double_Output, Ramp_Fault)
    := START_WHAT='Nominal_functioning';
END_TRANSITION
STEP Dummy11:
END_STEP
STEP Ramp_Range:
    RampRange_active(N);  // step action
END_STEP
TRANSITION FROM Ramp_Range TO Ramp_Range
    := TRUE;
END_TRANSITION
STEP Double_Output:
    Double_Output_active(N);  // step action
END_STEP
TRANSITION FROM Double_Output TO Double_Output
    := TRUE;
END_TRANSITION
STEP Ramp_Fault:
    Ramp_Fault_active(N);  // step action
END_STEP
TRANSITION FROM Ramp_Fault TO Ramp_Fault
    := TRUE;
END_TRANSITION
TRANSITION FROM Dummy11 TO MotorSlow
    := TRUE;
END_TRANSITION
STEP MotorSlow:
    MotorSlow_active(N);  // step action
    MotorSlow_exit(P0);  // exit action
END_STEP
TRANSITION FROM MotorSlow TO MotorFast
    := RampRange=FALSE;
END_TRANSITION
STEP MotorFast:
    MotorFast_active(N);  // step action
END_STEP
TRANSITION FROM MotorFast TO StopORGo
    := TRUE;
END_TRANSITION
STEP StopORGo:
    StopORGo_active(N);  // step action
END_STEP
TRANSITION FROM StopORGo TO MotorSlow
    := minni=TRUE;
END_TRANSITION
TRANSITION FROM BUSY TO Vel_Init
    := START_WHAT='Initialization';
END_TRANSITION
STEP Vel_Init:
    Vel_Init_active(N);  // step action
    Vel_Init_exit(P0);  // exit action
END_STEP
TRANSITION FROM Vel_Init TO READY
    := STOP;
END_TRANSITION

ACTION Double_Output_active:
//This two operation are done to copy the value of I_Vel and I_RampSensor into two new variables in order
//two use this value in another GA without violated the rules of the GA approach

I_Vel_2:=I_Vel;
I_RampSensor_2:=I_RampSensor;
END_ACTION

ACTION MotorSlow_active:
//We set a LOW SPEED until we are inside the RampRange of the floor where we have just stopped.
I_Vel:=FALSE;
END_ACTION

ACTION MotorSlow_exit:
//minni, whose meaning is well explained in block StopORGo, is reset to FALSE because we are going back to a FAST situation
//and we will need minni to detect if we need to SLOW DOWN again the motor.

minni:=FALSE;
END_ACTION

ACTION MotorFast_active:
//If we are not in the RampRange of the next destination (or if we are moving away from a stop, but we still are in the
//RampRange that stop), the VEL must be FAST.
I_Vel:=TRUE;
bunny:=FALSE; //The value of bunny, whose meaning is well explained in block StopORGo, is reset in order to use it properly
//in the next block
END_ACTION

ACTION StopORGo_active:
//SANDWICH PROBLEM 

//The lift is slowed down only when it meets the rampsensor of the destination floor.
//Minni is set to true if the lift has to slow down.
//Bunny is used to calculate the next velocity only once per RampRange (so minni is updated maximum once per RampRange). 
//This is useful because when the lift  reaches the deck sensor and the GVL.Destination is the following floor, 
//minni would become true even if we haven't reached yet the destination floor. 
//bunny returns false everytime the lift goes outside the RampRange, so bunny waits the next ramprange to 
//become true again.

//So when minni=TRUE, the next transition is satisfied and we can go in the block MotorSlow.

IF RampRange=TRUE THEN
	IF ((I_go_up=TRUE AND GVL.Destination-GVL.Current=1)OR(I_go_up=FALSE AND GVL.Destination-GVL.Current=-1)) AND bunny=FALSE THEN
	minni:=TRUE;
	END_IF
	bunny:=TRUE;
END_IF
IF RampRange=FALSE THEN
	bunny:=FALSE;
END_IF
END_ACTION

ACTION RampRange_active:
// This block calculates if we are inside or outside the two ramp sensors around the deck sensor of a floor.
//We implent the variable pluto because the turning on of the rampsensor can last more then a PLC cycle
//(we don't know the duration  of the signal), so thanks to pluto we can avoid counting twice the change
//of RampRange value.

//RampRange changes its value only when a RampSensor becomes true, whereas it is not affected when RampSensor
//becomes false.


IF I_RampSensor=TRUE AND RampRange=TRUE AND pluto=FALSE THEN
	pluto:=TRUE;
	RampRange:=FALSE;
END_IF
IF I_RampSensor=TRUE AND RampRange=FALSE AND pluto=FALSE THEN
	RampRange:=TRUE;
	pluto:=TRUE;
END_IF
IF I_RampSensor=FALSE THEN
	pluto:=FALSE;
END_IF
END_ACTION

ACTION Init_active:
STATE:='Init';
//All the variable useful in the nominal_functioning are initialiazed correctly here
RampRange:=TRUE;
pluto:=FALSE;
minni:=FALSE;
bunny:=FALSE;

EndInit:=TRUE;
END_ACTION

ACTION READY_active:
STATE:= 'READY';
END_ACTION

ACTION BUSY_active:
STATE:='BUSY';
END_ACTION

ACTION Vel_Init_active:
//Vel is set to LOW SPEED as requested by the initialization procedure
I_Vel:=FALSE;

Init_Done:=TRUE; //it comunicates to the policy that the initialization is completed
END_ACTION

ACTION Vel_Init_exit:
Init_Done:=FALSE;
END_ACTION

ACTION Ramp_Fault_active:
(*This block tries to detect a Ramp Fault. The management of this fault, actually is done by the Policy in the blocks
ARRAI and Delete_Array. When a broken ramp sensor is detected then some stops are not possible anymore if we do not
want to slow down permanently the lift (easier solution). The stops that cannot be performed are the once where the
broken ramp sensor don't allow us to slow down in time to stop at that floor. In this case the lift goes to the closest 
floor (according to the direction that it had) and then goes back to the previous floor coming now from the opposite
direction where the ramp sensor works. Special situation happen when the elevator is called at the floor X (the has to 
be reached going thru the broken sensor positioned just before the floor X) and just from one or more lower floor 
(considering in this example that to reach X the elevator is going up; same consideration, but mirrored can be done 
if we are going down), in this case the elevator does not go to X+1, but directly to X-2 (consider that also X-1 is not
servable if the elevator goes down) in order to optimize the movements. A throw back of this implementation is that, 
if there were a call from X-1 this got lost when destionation is X*)


//NRST and NRST_2 are used to count I_RampSensor only once when it is activated. The initial values for NRST 
//and NRST_2 are FALSE.

//Whenever I_RampSensor becomes TRUE, NRST is set as TRUE. This is excuted only for the first cycle for which
//I_RampSensor is TRUE because possible double counting of the same signal are stopped by NRST_2, that some 
//lines down is set as TRUE.
IF I_RampSensor AND NRST_2=FALSE THEN
	NRST:=TRUE; //NRST stands for Not Ramp Sensor Twice
END_IF

//When I_RampSensor gets FALSE we reset the values of NRST and NRST_2 to be ready for the next time in which
//I_RampSensor becomes TRUE.
IF I_RampSensor=FALSE THEN
	NRST:=FALSE;
	NRST_2:=FALSE;
END_IF


//When we have detected the first turning TRUE of I_RampSensor, we have NRST=TRUE, so we update the variable
//count_ramp. This variable keeps the count of how many ramp sensors are met without meeting a DeckSensor.
//This little block is excuted only once per meeting with a RampSensor, indeed the first time we excute it we also 
//set NRST_2:=TRUE and NRST:=FALSE; this will block the first IF of this code as well as this IF itself. We can 
//excute again this two IF only after a reset of NRST and NRST_2, that happens when I_RampSensor gets FALSE.
IF NRST THEN 
	count_ramp:=count_ramp+1;
	NRST_2:=TRUE;
	NRST:=FALSE; 
END_IF

(*When a DeckSensor is met and count_ramp is equal to 1, it means that there is a broken RampSensor. To inform the
policy of this discoverage we use the variable I_FaultRampAlarm that will remain TRUE. Moreover also the variable
I_RampAlarm is created, and this one remains TRUE only until the lift leaves the DeckSensor. This variable is then
used by the policy in the blocks ARRAI and DeleteArray.*)
IF count_ramp=1 AND I_DeckSensor THEN
	I_FaultRampAlarm:=TRUE;
	I_RampAlarm:=TRUE;
END_IF

(*The variable 'pip' is helpful to execute the next IF a cycle after the previous IF. Indeed if these two blocks would
be performed in the same moment they would conflict*)
IF I_DeckSensor AND pip=FALSE THEN
	pip:=TRUE;
END_IF

(*Once that the lift has leaved the DeckSensor the variables can be reset*)
IF I_DeckSensor=FALSE AND pip THEN
	pip:=FALSE;
	count_ramp:=0;
	RampRange:=TRUE;
	I_RampAlarm:=FALSE;
END_IF
END_ACTION

END_FUNCTION_BLOCK

// Device/Application/Visualization
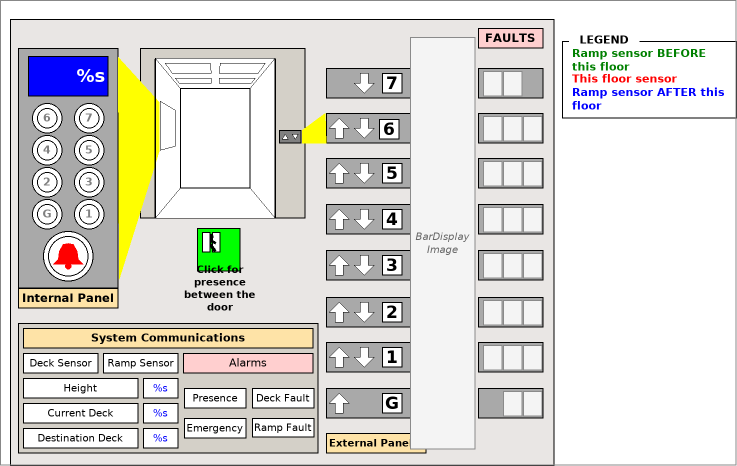
VISUALIZATION Visualization  // 737x466
    Rectangle (10,19 544x447)
    Rectangle (197,228 43x43), colour toggle: GVL.Presence
    Rectangle (18,323 300x130)
    Rectangle (326,433 100x20), "External Panels"
    Rectangle (326,342 100x30)
    Rectangle (382,347 20x20), "1"
    Polygon (354,357) (360,357) (360,347) (368,347) (368,357) (374,357) (364,367), colour toggle: GVL.DownDeck1Vis
        tap GVL.DownDeck1
    Polygon (329,357) (335,357) (335,367) (343,367) (343,357) (349,357) (339,347), colour toggle: GVL.UpDeck1Vis
        tap GVL.UpDeck1
    Rectangle (326,297 100x30)
    Rectangle (382,302 20x20), "2"
    Polygon (354,312) (360,312) (360,302) (368,302) (368,312) (374,312) (364,322), colour toggle: GVL.DownDeck2Vis
        tap GVL.DownDeck2
    Polygon (329,312) (335,312) (335,322) (343,322) (343,312) (349,312) (339,302), colour toggle: GVL.UpDeck2Vis
        tap GVL.UpDeck2
    Rectangle (326,250 100x30)
    Rectangle (382,255 20x20), "3"
    Polygon (354,265) (360,265) (360,255) (368,255) (368,265) (374,265) (364,275), colour toggle: GVL.DownDeck3Vis
        tap GVL.DownDeck3
    Polygon (329,265) (335,265) (335,275) (343,275) (343,265) (349,265) (339,255), colour toggle: GVL.UpDeck3Vis
        tap GVL.UpDeck3
    Rectangle (326,204 100x30)
    Rectangle (382,209 20x20), "4"
    Polygon (354,219) (360,219) (360,209) (368,209) (368,219) (374,219) (364,229), colour toggle: GVL.DownDeck4Vis
        tap GVL.DownDeck4
    Polygon (329,219) (335,219) (335,229) (343,229) (343,219) (349,219) (339,209), colour toggle: GVL.UpDeck4Vis
        tap GVL.UpDeck4
    Rectangle (326,158 100x30)
    Rectangle (382,163 20x20), "5"
    Polygon (354,173) (360,173) (360,163) (368,163) (368,173) (374,173) (364,183), colour toggle: GVL.DownDeck5Vis
        tap GVL.DownDeck5
    Polygon (329,173) (335,173) (335,183) (343,183) (343,173) (349,173) (339,163), colour toggle: GVL.UpDeck5Vis
        tap GVL.UpDeck5
    Rectangle (326,113 100x30)
    Rectangle (379,119 20x20), "6"
    Polygon (354,128) (360,128) (360,118) (368,118) (368,128) (374,128) (364,138), colour toggle: GVL.DownDeck6Vis
        tap GVL.DownDeck6
    Polygon (329,128) (335,128) (335,138) (343,138) (343,128) (349,128) (339,118), colour toggle: GVL.UpDeck6Vis
        tap GVL.UpDeck6
    Rectangle (326,68 100x30)
    Rectangle (382,73 20x20), "7"
    Polygon (354,83) (360,83) (360,73) (368,73) (368,83) (374,83) (364,93), colour toggle: GVL.DownDeck7Vis
        tap GVL.DownDeck7
    Rectangle (326,388 100x30)
    Rectangle (382,393 20x20), "G"
    Polygon (329,403) (335,403) (335,413) (343,413) (343,403) (349,403) (339,393), colour toggle: GVL.UpDeckGVis
        tap GVL.UpDeckG
    RoundedRectangle (18,48 100x240)
    Rectangle (18,288 100x20), "Internal Panel"
    Ellipse (74,199 30x30), colour toggle: GVL.P1Vis
    Ellipse (79,204 20x20), "1"
        tap GVL.P1
    Ellipse (32,199 30x30), colour toggle: GVL.PGVis
    Ellipse (37,204 20x20), "G"
        tap GVL.PG
    Ellipse (74,167 30x30), colour toggle: GVL.P3Vis
    Ellipse (79,172 20x20), "3"
        tap GVL.P3
    Ellipse (32,167 30x30), colour toggle: GVL.P2Vis
    Ellipse (37,172 20x20), "2"
        tap GVL.P2
    Ellipse (74,135 30x30), colour toggle: GVL.P5Vis
    Ellipse (79,140 20x20), "5"
        tap GVL.P5
    Ellipse (32,135 30x30), colour toggle: GVL.P4Vis
    Ellipse (37,140 20x20), "4"
        tap GVL.P4
    Ellipse (74,103 30x30), colour toggle: GVL.P7Vis
    Ellipse (79,108 20x20), "7"
        tap GVL.P7
    Ellipse (32,103 30x30), colour toggle: GVL.P6Vis
    Ellipse (37,108 20x20), "6"
        tap GVL.P6
    Rectangle (28,56 80x40), "%s", text variable: GVL.Destination
    Ellipse (43,231 50x50), tooltip "EMERGENCY", colour toggle: GVL.Emergency
    Group (48,236 40x40)
        toggle GVL.Emergency
        Ellipse (0,0 40x40), tooltip "EMERGENCY"
        Polygon (5,28) (10,23) (11,15) (15,8) (20,7) (25,8) (29,15) (30,23) (35,28)
        Ellipse (17,27 6x6)
    Polygon (35,72) (45,62) (55,72), colour toggle: GVL.Motor_on AND GVL.Up
    Polygon (35,80) (45,90) (55,80), colour toggle: GVL.Motor_on AND NOT GVL.Up
    Group (140,48 165x170)
        Rectangle (0,0 165x170)
        Rectangle (15,10 120x160)
        Polygon (40,40) (15,10) (135,10) (110,40)
        Rectangle (40,40 70x100)
        Polygon (15,170) (40,140) (110,140) (135,170)
        Polygon (20,102) (20,53) (35,62) (35,98)
        Polygon (79,35) (79,30) (115,30) (111,35)
        Polygon (39,35) (35,30) (71,30) (71,35)
        Polygon (32,25) (25,15) (70,15) (71,25)
        Polygon (79,25) (80,15) (125,15) (118,25)
        Group (139,82 22x13)
            Rectangle (0,0 22x13)
            Polygon (3,9) (6,4) (9,9)
            Polygon (13,4) (16,9) (19,4)
    BarDisplayImage (410,37 65x412), value: GVL.Height, style: BarDisplayImage-Gray, scale format: %.0f, scale -20..160
        p3451962224: VisuNativeControl.IP_Offline.Browser
    Rectangle (478,68 65x30)
    Rectangle (478,342 65x30)
    Rectangle (478,297 65x30)
    Rectangle (478,250 65x30)
    Rectangle (478,204 65x30)
    Rectangle (478,158 65x30)
    Rectangle (478,113 65x30)
    Rectangle (478,388 65x30)
    RockerSwitch (483,345 19x25), variable: GVL.Ramp1Down, behaviour: TOGGLE, style: Switch-RockerSwitch-Green
    RockerSwitch (503,345 19x25), variable: GVL.Sensor1, behaviour: TOGGLE, style: Switch-RockerSwitch-Red
    RockerSwitch (523,345 19x25), variable: GVL.Ramp1Up, behaviour: TOGGLE, style: Switch-RockerSwitch-Blue
    RockerSwitch (483,300 19x25), variable: GVL.Ramp2Down, behaviour: TOGGLE, style: Switch-RockerSwitch-Green
    RockerSwitch (503,300 19x25), variable: GVL.Sensor2, behaviour: TOGGLE, style: Switch-RockerSwitch-Red
    RockerSwitch (523,300 19x25), variable: GVL.Ramp2Up, behaviour: TOGGLE, style: Switch-RockerSwitch-Blue
    RockerSwitch (483,253 19x25), variable: GVL.Ramp3Down, behaviour: TOGGLE, style: Switch-RockerSwitch-Green
    RockerSwitch (503,253 19x25), variable: GVL.Sensor3, behaviour: TOGGLE, style: Switch-RockerSwitch-Red
    RockerSwitch (523,253 19x25), variable: GVL.Ramp3Up, behaviour: TOGGLE, style: Switch-RockerSwitch-Blue
    RockerSwitch (483,207 19x25), variable: GVL.Ramp4Down, behaviour: TOGGLE, style: Switch-RockerSwitch-Green
    RockerSwitch (503,207 19x25), variable: GVL.Sensor4, behaviour: TOGGLE, style: Switch-RockerSwitch-Red
    RockerSwitch (523,207 19x25), variable: GVL.Ramp4Up, behaviour: TOGGLE, style: Switch-RockerSwitch-Blue
    RockerSwitch (483,161 19x25), variable: GVL.Ramp5Down, behaviour: TOGGLE, style: Switch-RockerSwitch-Green
    RockerSwitch (503,161 19x25), variable: GVL.Sensor5, behaviour: TOGGLE, style: Switch-RockerSwitch-Red
    RockerSwitch (523,161 19x25), variable: GVL.Ramp5Up, behaviour: TOGGLE, style: Switch-RockerSwitch-Blue
    RockerSwitch (483,116 19x25), variable: GVL.Ramp6Down, behaviour: TOGGLE, style: Switch-RockerSwitch-Green
    RockerSwitch (503,116 19x25), variable: GVL.Sensor6, behaviour: TOGGLE, style: Switch-RockerSwitch-Red
    RockerSwitch (523,116 19x25), variable: GVL.Ramp6Up, behaviour: TOGGLE, style: Switch-RockerSwitch-Blue
    RockerSwitch (483,71 19x25), variable: GVL.Ramp7Down, behaviour: TOGGLE, style: Switch-RockerSwitch-Green
    RockerSwitch (503,71 19x25), variable: GVL.Sensor7, behaviour: TOGGLE, style: Switch-RockerSwitch-Red
    RockerSwitch (503,391 19x25), variable: GVL.SensorG, behaviour: TOGGLE, style: Switch-RockerSwitch-Red
    RockerSwitch (523,391 19x25), variable: GVL.RampGUp, behaviour: TOGGLE, style: Switch-RockerSwitch-Blue
    Rectangle (478,28 65x20), "FAULTS"
    Polygon (302,130) (325,113) (326,143) (302,143), invisible if: (GVL.Closing OR GVL.Opening) OR GVL.Closed
    Polygon (118,57) (159,102) (159,151) (119,279), invisible if: (GVL.Closing OR GVL.Opening) OR GVL.Closed
    Rectangle (155,58 0x160)
        p3528305787: GVL.Door
    Rectangle (275,58 0x160)
        p3528305787: -GVL.Door
    Rectangle (23,328 290x20), "System Communications"
    Rectangle (183,353 130x20), "Alarms"
    Rectangle (23,353 75x20), "Deck Sensor", colour toggle: GVL.DeckSensor
    Rectangle (143,378 35x20), "%s", text variable: GVL.Height
    Rectangle (184,388 62x20), "Presence", colour toggle: GVL.Presence
    Rectangle (103,353 75x20), "Ramp Sensor", colour toggle: GVL.RampSensor
    Rectangle (143,403 35x20), "%s", text variable: GVL.Current
    Rectangle (143,428 35x20), "%s", text variable: GVL.Destination
    Rectangle (252,388 62x20), "Deck Fault", colour toggle: GVL.FaultSensorAlarm
    Rectangle (184,418 62x20), "Emergency", colour toggle: GVL.EmergencyVis
    Rectangle (252,418 62x19), "Ramp Fault", colour toggle: GVL.FaultRampAlarm
    Rectangle (23,378 115x20), "Height"
    Rectangle (23,403 115x20), "Current Deck"
    Rectangle (23,428 115x20), "Destination Deck"
    Group (562,25 175x93)
        Rectangle (0,16 175x77)
        Rectangle (7,39 160x30), "This floor sensor"
        Rectangle (7,59 160x30), "Ramp sensor AFTER this floor"
        Rectangle (7,0 70x30), "LEGEND"
        Rectangle (7,20 160x30), "Ramp sensor BEFORE this floor"
    Group (202,232 33x34)
        toggle GVL.Presence
        Rectangle (10,0 8x20)
        Polygon (5,10) (12,20) (14,18) (5,6)
        Ellipse (6,2 5x5)
        Polygon (4,8) (13,12) (14,10) (4,4)
        Rectangle (0,0 8x20)
    Rectangle (169,273 102x31), "Click for presence between the door"
END_VISUALIZATION
